	CODE_START := CODE_START + 1;
	// pull out the parameters
	SCREW_PARAMETERS[NS_PITCH] := STRING_TO_REAL(MID(GPS_PNEZD_D, 3, CODE_START));
	SCREW_PARAMS_CUSTOM[0].NS_PITCH := STRING_TO_SINT(MID(GPS_PNEZD_D, 3, CODE_START));
	CODE_START := CODE_START + 3;
	SCREW_PARAMETERS[SCREW_LENGTH] := STRING_TO_REAL(MID(GPS_PNEZD_D, 3, CODE_START));
	SCREW_PARAMS_CUSTOM[0].SCREW_LENGTH := STRING_TO_UINT(MID(GPS_PNEZD_D, 3, CODE_START));
	CODE_START := CODE_START + 3;
	SCREW_PARAMETERS[TRUSS_VERT_ANGLE] := STRING_TO_REAL(MID(GPS_PNEZD_D, 2, CODE_START));
	SCREW_PARAMS_CUSTOM[0].TRUSS_VERT_ANGLE := STRING_TO_USINT(MID(GPS_PNEZD_D, 2, CODE_START));
	CODE_START := CODE_START + 2;
	IF MID(GPS_PNEZD_D, 2, CODE_START) = 'ZZ' OR MID(GPS_PNEZD_D, 2, CODE_START) = 'zz' THEN
		SCREW_PARAMETERS[THIRD_LEG_VERT_ANGLE] := NA;
		SCREW_PARAMS_CUSTOM[0].THIRD_LEG_VERT_ANGLE := TO_USINT(NA);
	ELSE
		SCREW_PARAMETERS[THIRD_LEG_VERT_ANGLE] := STRING_TO_REAL(MID(GPS_PNEZD_D, 2, CODE_START));
		SCREW_PARAMS_CUSTOM[0].THIRD_LEG_VERT_ANGLE := STRING_TO_USINT(MID(GPS_PNEZD_D, 2, CODE_START));
	END_IF
	CODE_START := CODE_START + 2;
	SCREW_PARAMETERS[EMBED_LENGTH] := STRING_TO_REAL(MID(GPS_PNEZD_D, 3, CODE_START));
	SCREW_PARAMS_CUSTOM[0].EMBED_LENGTH := STRING_TO_USINT(MID(GPS_PNEZD_D, 3, CODE_START));
	CODE_START := CODE_START + 3;
	IF MID(GPS_PNEZD_D, 2, CODE_START) = 'ZZ' OR MID(GPS_PNEZD_D, 2, CODE_START) = 'zz' THEN
		SCREW_PARAMETERS[IE_MIN_HAMMER] := NA;
		SCREW_PARAMS_CUSTOM[0].IE_MIN_HAMMER := TO_USINT(NA);
	ELSE
		SCREW_PARAMETERS[IE_MIN_HAMMER] := STRING_TO_REAL(MID(GPS_PNEZD_D, 2, CODE_START));
		SCREW_PARAMS_CUSTOM[0].IE_MIN_HAMMER := STRING_TO_USINT(MID(GPS_PNEZD_D, 2, CODE_START));
	END_IF
	CODE_START := CODE_START + 2;
	IF MID(GPS_PNEZD_D, 2, CODE_START) = 'ZZ' OR MID(GPS_PNEZD_D, 2, CODE_START) = 'zz' THEN
		SCREW_PARAMETERS[IE_MIN_EMBED] := NA;
		SCREW_PARAMS_CUSTOM[0].IE_MIN_EMBED := TO_USINT(NA);
	ELSE
		SCREW_PARAMETERS[IE_MIN_EMBED] := STRING_TO_REAL(MID(GPS_PNEZD_D, 2, CODE_START));
		SCREW_PARAMS_CUSTOM[0].IE_MIN_EMBED := STRING_TO_USINT(MID(GPS_PNEZD_D, 2, CODE_START));
	END_IF
	CODE_START := CODE_START + 2;
	DecodePnezD := TRUE;
	//SCREW_PARAMETERS[TRUSS_TYPE] := AsciiToReal(MID(GPS_PNEZD_D, 1, CODE_START));
	(*
	IF MID(GPS_PNEZD_D, 1, CODE_START) = TRUSS_CODES[] OR MID(GPS_PNEZD_D, 1, CODE_START) = 'i' THEN
		SCREW_PARAMETERS[TRUSS_TYPE] := 0;
	ELSIF MID(GPS_PNEZD_D, 1, CODE_START) = 'E' OR MID(GPS_PNEZD_D, 1, CODE_START) = 'e' THEN
		SCREW_PARAMETERS[TRUSS_TYPE] := 2;
	ELSIF MID(GPS_PNEZD_D, 1, CODE_START) = 'C' OR MID(GPS_PNEZD_D, 1, CODE_START) = 'c' THEN
		SCREW_PARAMETERS[TRUSS_TYPE] := 1;
	ELSE
		DecodePnezD := FALSE;
	END_IF*)

END_FUNCTION

// StandardPLC/Application/POUs/Utilities/Conversions/AsciiToReal
FUNCTION AsciiToReal : REAL
VAR_INPUT
	CHAR: STRING(1);
END_VAR
VAR
	pBYTE: POINTER TO BYTE;
END_VAR

pBYTE := ADR(CHAR);
AsciiToReal := pBYTE^;

END_FUNCTION

// StandardPLC/Application/POUs/Test_PRGs/DynamicList
(* This list self-populates with new values until the max size is reached.
eg, if a new screw size is added, it will automatically add it to the list and start counting that size screw.
*)

PROGRAM DynamicList 
VAR
	// function vars
	i: USINT := 0;
	
	// sim vars
	init: BOOL := TRUE;
	pnezDlast: STRING(64) := '';
	// system vars
	SCREW_COUNT_ORDER: ARRAY [1..SCREW_LENGTHS_COUNT] OF UDINT := [SCREW_LENGTHS_COUNT(0)];
	
	
END_VAR

IF init OR (pnezDlast <> GPS_PNEZD_D) THEN
	init := FALSE;
	pnezDlast := GPS_PNEZD_D;
	
	FOR i := 1 TO SCREW_LENGTHS_COUNT DO
		IF TO_UINT(SCREW_COUNT[1,i]) = TO_UINT(SCREW_PARAMETERS[SCREW_LENGTH]) THEN
			SCREW_COUNT[2,i] := SCREW_COUNT[2,i] + 1;
			EXIT;
		ELSIF TO_UINT(SCREW_COUNT[1,i]) = 0 THEN
			SCREW_COUNT[1,i] := TO_UINT(SCREW_PARAMETERS[SCREW_LENGTH]);
			SCREW_COUNT[2,i] := 1;
			// *** organize list
			WHILE i > 1 DO
				IF SCREW_COUNT[1,i] < SCREW_COUNT[1,i - 1] THEN
					SCREW_COUNT[1,i] := SCREW_COUNT[1,i - 1];
					SCREW_COUNT[2,i] := SCREW_COUNT[2,i - 1];
					SCREW_COUNT[1,i-1] := TO_UINT(SCREW_PARAMETERS[SCREW_LENGTH]);
					SCREW_COUNT[2,i-1] := 1;
				END_IF
				i := i - 1;
			END_WHILE
			EXIT;
			// ^^^
		END_IF
	END_FOR	
END_IF

END_PROGRAM

// StandardPLC/Application/POUs/Test_PRGs/Arrays
PROGRAM Arrays
VAR
	Init: BOOL := TRUE;
	TEST_1: ARRAY [0..20] OF UINT := [15,20(0)]; // first position indicates number of used slots
	TEST_2: ARRAY [3..9] OF BOOL := [7(0)];	
	TEST_3: ARRAY [0..20] OF UINT := [21(0)];
	LOWER_BOUND_TEST_1: USINT := 0;
	LOWER_BOUND_TEST_2: USINT := 0;
	UPPER_BOUND_TEST_1: USINT := 0;
	UPPER_BOUND_TEST_2: USINT := 0;
	LENGTH_TEST_1: USINT := 0;
	LENGTH_TEST_2: USINT := 0;
	SIZE_OF_TEST_1: UINT := 0;
	SIZE_OF_TEST_2: UINT := 0;
	i: UINT := 0;
	j: UINT := 0;
	Timeout_Index: UINT := 0;
END_VAR

IF Init THEN
	Init := FALSE;
	Timeout_Index := 1;
	//LOWER_BOUND_TEST_1 := TO_USINT(LOWER_BOUND(TEST_1, 2));
	//LOWER_BOUND_TEST_2 := TO_USINT(LOWER_BOUND(TEST_2, 1));
	//UPPER_BOUND_TEST_1 := TO_USINT(UpperBoundBool(TEST_1));
	UPPER_BOUND_TEST_2 := TO_USINT(UpperBoundBool(TEST_2));
	SIZE_OF_TEST_1 := SIZEOF(TEST_1);
	SIZE_OF_TEST_2 := SIZEOF(TEST_2);

END_IF
Timeout_Index := Timeout_Index + 1;
IF Timeout_Index <= 200 THEN
	FOR i := 1 TO TEST_1[0] DO
		TEST_1[i] := TEST_1[i] + i;
	END_FOR
ELSIF Timeout_Index = 300 THEN
	TEST_3 := TEST_1;
	
END_IF

END_PROGRAM

// StandardPLC/Application/POUs/Utilities/UpperBoundBool
FUNCTION UpperBoundBool : UINT
VAR_IN_OUT
	INPUT_ARRAY : ARRAY[*] OF BOOL;
END_VAR
VAR_INPUT
	
END_VAR
VAR
END_VAR

UpperBoundBool := TO_UINT(UPPER_BOUND(INPUT_ARRAY, 1));

END_FUNCTION

// Project Information/GetCompany
// This function has been automatically generated from the project information.
{attribute 'signature_flag' := '1073741824'}
{attribute 'register_in_runtime'}
FUNCTION GetCompany : WSTRING
VAR_INPUT
	
END_VAR

GetCompany := "ifm electronic";

END_FUNCTION

// Project Information/GetTitle
// This function has been automatically generated from the project information.
{attribute 'signature_flag' := '1073741824'}
{attribute 'register_in_runtime'}
FUNCTION GetTitle : WSTRING
VAR_INPUT
	
END_VAR

GetTitle := "ifmCR711S_TemplateProject";

END_FUNCTION

// Project Information/GetVersion
// This function has been automatically generated from the project information.
{attribute 'signature_flag' := '1073741824'}
{attribute 'register_in_runtime'}
FUNCTION GetVersion : VERSION
VAR_INPUT
	
END_VAR

GetVersion.uiMajor := 2;
GetVersion.uiMinor := 4;
GetVersion.uiServicePack := 15;
GetVersion.uiPatch := 0;

END_FUNCTION

// Project Information/GetTextProperty
// This function has been automatically generated from the project information.
{attribute 'signature_flag' := '1073741824'}
{attribute 'register_in_runtime'}
FUNCTION GetTextProperty : WSTRING
VAR_INPUT
	stKey: WSTRING;
END_VAR

IF stKey = "Company" THEN
	GetTextProperty := "ifm electronic";
ELSIF stKey = "Description" THEN
	GetTextProperty := "Project template with CR711S configured 2.25MByte Standard 2.25MByte Safety";
ELSIF stKey = "Project" THEN
	GetTextProperty := "experiment_with_CoDeSys_sp16";
ELSIF stKey = "Title" THEN
	GetTextProperty := "ifmCR711S_TemplateProject";
ELSE
	GetTextProperty := "";
END_IF

END_FUNCTION

// Project Information/GetTextProperty2
// This function has been automatically generated from the project information.
{attribute 'signature_flag' := '1073741824'}
{attribute 'register_in_runtime'}
FUNCTION GetTextProperty2 : POINTER TO WSTRING
VAR_INPUT
	stKey: WSTRING;
END_VAR

IF stKey = "Company" THEN
	GetTextProperty2 := ADR("ifm electronic");
ELSIF stKey = "Description" THEN
	GetTextProperty2 := ADR("Project template with CR711S configured 2.25MByte Standard 2.25MByte Safety");
ELSIF stKey = "Project" THEN
	GetTextProperty2 := ADR("experiment_with_CoDeSys_sp16");
ELSIF stKey = "Title" THEN
	GetTextProperty2 := ADR("ifmCR711S_TemplateProject");
ELSE
	GetTextProperty2 := ADR("");
END_IF

END_FUNCTION

// Project Information/GetNumberProperty
// This function has been automatically generated from the project information.
{attribute 'signature_flag' := '1073741824'}
{attribute 'register_in_runtime'}
FUNCTION GetNumberProperty : DINT
VAR_INPUT
	stKey: WSTRING;
END_VAR

GetNumberProperty := 0;

END_FUNCTION

// Project Information/GetBooleanProperty
// This function has been automatically generated from the project information.
{attribute 'signature_flag' := '1073741824'}
{attribute 'register_in_runtime'}
FUNCTION GetBooleanProperty : BOOL
VAR_INPUT
	stKey: WSTRING;
END_VAR

IF stKey = "Released" THEN
	GetBooleanProperty := FALSE;
ELSE
	GetBooleanProperty := FALSE;
END_IF

END_FUNCTION

// Project Information/GetVersionProperty
// This function has been automatically generated from the project information.
{attribute 'signature_flag' := '1073741824'}
{attribute 'register_in_runtime'}
FUNCTION GetVersionProperty : VERSION
VAR_INPUT
	stKey: WSTRING;
END_VAR

IF stKey = "Version" THEN
	GetVersionProperty.uiMajor := 2;
	GetVersionProperty.uiMinor := 4;
	GetVersionProperty.uiServicePack := 15;
	GetVersionProperty.uiPatch := 0;
ELSE
	GetVersionProperty.uiMajor := 0;
	GetVersionProperty.uiMinor := 0;
	GetVersionProperty.uiServicePack := 0;
	GetVersionProperty.uiPatch := 0;
END_IF

END_FUNCTION

// StandardPLC/Application/POUs/Utilities/Conversions/pSQR
FUNCTION pSqr : POINTER TO REAL
VAR_INPUT
	Num: REAL;
	
END_VAR
VAR
		SqrVal: LREAL;
END_VAR


SqrVal := EXPT(Num, 2);
pSqr := ADR (SqrVal);

END_FUNCTION

// StandardPLC/Application/POUs/Utilities/Conversions/SqrReals
FUNCTION SqrReals : REAL
VAR_INPUT
	Num: REAL;

END_VAR
VAR
END_VAR

SqrReals := to_real(EXPT(Num,2));

END_FUNCTION

// StandardPLC/Application/POUs/ConvertDiag
FUNCTION_BLOCK ConvertDiag
VAR_INPUT
	ifmDiag: ifmTYPES.DIAG_INFO;
END_VAR
VAR_OUTPUT
	s_Diag: STRING;
END_VAR
VAR
	i_Diag: Diag;
END_VAR

(* input is TO_INT(ifm ediag's name)
create a diag enum with this as the number
convert diag to string with to_string*)

i_Diag := TO_INT(ifmDiag);
s_Diag := TO_STRING(i_Diag);

END_FUNCTION_BLOCK

// StandardPLC/Application/POUs/ConvDiag
FUNCTION ConvDiag : STRING
VAR_INPUT
		ifmDiag: ifmTYPES.DIAG_INFO;
END_VAR
VAR
	i_diag: diag;
END_VAR



i_diag := TO_INT(ifmDiag);
ConvDiag := TO_STRING(i_diag);

END_FUNCTION

// StandardPLC/Application/POUs/Checksum
FUNCTION Checksum : UINT

VAR_INPUT
	FILE_PTR: POINTER TO BYTE; // pointer to beginning of memory block/file to be checked
	FILE_LENGTH: UINT; // # of bytes in file
END_VAR

VAR
	INDEX: INT; // loop index
	SUM: UINT := 0; // sum of 1's in file
	
END_VAR

FILE_LENGTH := MAX(1,FILE_LENGTH);

FOR INDEX := 1 TO TO_INT(FILE_LENGTH) DO
	SUM := SUM + TO_UINT(FILE_PTR^);
	FILE_PTR := FILE_PTR + 1;
END_FOR

Checksum := SUM;

END_FUNCTION

// StandardPLC/Application/POUs/Utilities/MemBlockLength
FUNCTION MemBlockLength : UINT
VAR_INPUT
	PTR_START: POINTER TO BYTE;
	PTR_END: POINTER TO BYTE;
	
END_VAR
VAR
	FILE_LENGTH: DWORD := 0;
END_VAR


FILE_LENGTH := MAX(1, ABS(PTR_END - PTR_START));
MemBlockLength := TO_UINT(FILE_LENGTH);

END_FUNCTION

// StandardPLC/Application/POUs/Checksum_wLength
FUNCTION Checksum_wLength : UINT

VAR_INPUT
	FILE_BEGIN_PTR: POINTER TO BYTE; // pointer to beginning of memory block/file to be checked
	FILE_END_PTR: POINTER TO BYTE; // pointer to end of memory block/file to be checked
END_VAR

VAR
	INDEX: INT := 0; // loop index
	SUM: UINT := 0; // sum of 1's in file
	
	FILE_LENGTH: UINT := 0;
END_VAR


FILE_LENGTH := MemBlockLength(FILE_BEGIN_PTR, FILE_END_PTR);
FILE_LENGTH := MAX(1,FILE_LENGTH);

FOR INDEX := 1 TO TO_INT(FILE_LENGTH) DO
	SUM := SUM + TO_UINT(FILE_BEGIN_PTR^);
	FILE_BEGIN_PTR := FILE_BEGIN_PTR + 1;
END_FOR

Checksum_wLength := SUM;

END_FUNCTION

// StandardPLC/Application/POUs/Utilities/Conversions/ArrayOfBytesToLWORD
FUNCTION ArrayOfBytesToLWORD : LWORD // not tested
VAR_INPUT
	ARRAY_SIZE: INT :=4; // accept arrays of 2 - 8 BYTES
	LITTLE_ENDIAN: BOOL := TRUE;
END_VAR
VAR_IN_OUT
	BYTE_ARRAY: ARRAY [*] OF BYTE;
END_VAR
VAR
	i: INT :=0;
	dataLWORD: LWORD :=0;
	BArray: ARRAY [0..8] OF BYTE := [0,0,0,0,0,0,0,0];
	
END_VAR

// concat array of bytes into LWORD
// rearrange for endianness
IF LITTLE_ENDIAN THEN
	dataLWORD :=  SHL(TO_LWORD(BArray[0]),8) OR BArray[1];
	FOR i := 0 TO ARRAY_SIZE - 1 DO
		BArray[ARRAY_SIZE - i - 1] := BYTE_ARRAY[i];
	END_FOR
ELSE
	dataLWORD := BArray[1] OR SHL(TO_LWORD(BArray[0]),8);
	FOR i := 0 TO ARRAY_SIZE - 1 DO
		BArray[i] := BYTE_ARRAY[i];
	END_FOR
END_IF

// pack arranged array into LWORD
dataLWORD :=  SHL(TO_LWORD(BArray[0]),8) OR BArray[1];
IF ARRAY_SIZE > 2 THEN
	FOR i := 2 TO ARRAY_SIZE - 1 DO
		dataLWORD := SHL(dataLWORD,8) OR BArray[i];
	END_FOR
END_IF

ArrayOfBytesToLWORD := dataLWORD;

END_FUNCTION

// StandardPLC/Application/POUs/Utilities/Conversions/ConvLWORDtoDecimal
FUNCTION ConvLWORDtoDecimal : REAL
VAR_INPUT
	BINARY: LWORD :=0;
	SCALE: REAL :=0;
	OFFSET: REAL :=0;
END_VAR
VAR
	DEC: INT := 0;
END_VAR

// input LWORD and output the scaled and offset decimal
//DEC := LWORD_TO_REAL (BINARY); // convert to INT first?
DEC := LWORD_TO_INT (BINARY);
ConvLWORDtoDecimal := INT_TO_REAL(DEC) * SCALE + OFFSET;

END_FUNCTION

// StandardPLC/Application/POUs/IsExtendedCAN
FUNCTION IsExtendedCAN : BOOL

VAR_INPUT
	MSG_ID: UDINT;
END_VAR
VAR
END_VAR

//IsExtendedCAN := (MSG_ID > 2047);

IsExtendedCAN := (len(TO_WORD(MSG_ID)) < 12);

END_FUNCTION

// StandardPLC/Application/POUs/getElapsedTime
FUNCTION_BLOCK getElapsedTime // not functional - just recorded ideas, didn't finish
VAR_INPUT
END_VAR
VAR_OUTPUT
END_VAR
VAR
	START: SysTime := 0;
	FINISH: SysTime := 0;
	INTERVAL: SysTime :=0;
	INTERVAL_SUM: SysTime :=0;
	INTERVAL_AVG: SysTime :=0;
END_VAR

// use systime to get microseconds or even nanoseconds for an event

SysTimeGetUs(START); // this is in the SysTime library; optional SysTimeGetNs.  assigns value to supplied variable 
// event occurs
SysTimeGetUs(FINISH);
INTERVAL := FINISH - START;

// if want to get an average add a count something like this:
(*
INTERVAL_SUM := INTERVAL_SUM + INTERVAL;
IF (COUNT MOD 1000 = 0) THEN
	INTERVAL_AVG := INTERVAL_SUM/1000;
	INTERVAL_SUM := 0;
END_IF
*)

END_FUNCTION_BLOCK

// StandardPLC/Application/POUs/Utilities/Conversions/REAL_TO_BYTE_ARRAY
FUNCTION_BLOCK REAL_TO_BYTE_ARRAY // take in a REAL and output an array of bytes
VAR_INPUT
END_VAR
VAR_OUTPUT
END_VAR
VAR
END_VAR

END_FUNCTION_BLOCK

// StandardPLC/Application/POUs/Utilities/Conversions/ArrayOfUsintsToLWORD
FUNCTION ArrayOfUsintsToLWORD : LWORD // not tested, may be a problem with this that crashes PLC
VAR_INPUT
	ARRAY_SIZE: INT :=4; // accept arrays of 2 - 8 BYTES
	LITTLE_ENDIAN: BOOL := TRUE;
END_VAR
VAR_IN_OUT
	BYTE_ARRAY: ARRAY [*] OF USINT;
END_VAR
VAR
	i: INT :=0;
	dataLWORD: LWORD :=0;
	BArray: ARRAY [0..8] OF BYTE := [0,0,0,0,0,0,0,0];
	
END_VAR

// concat array of bytes into LWORD
// rearrange for endianness

IF LITTLE_ENDIAN THEN
	dataLWORD :=  SHL(TO_LWORD(BArray[0]),8) OR BArray[1];
	FOR i := 0 TO ARRAY_SIZE - 1 DO
		BArray[ARRAY_SIZE - i - 1] := TO_BYTE(BYTE_ARRAY[i]);
	END_FOR
ELSE
	dataLWORD := BArray[1] OR SHL(TO_LWORD(BArray[0]),8);
	FOR i := 0 TO ARRAY_SIZE - 1 DO
		BArray[i] := TO_BYTE(BYTE_ARRAY[i]);
	END_FOR
END_IF

// pack arranged array into LWORD
dataLWORD :=  SHL(TO_LWORD(BArray[0]),8) OR BArray[1];
IF ARRAY_SIZE > 2 THEN
	FOR i := 2 TO ARRAY_SIZE - 1 DO
		dataLWORD := SHL(dataLWORD,8) OR BArray[i];
	END_FOR
END_IF

ArrayOfUsintsToLWORD := dataLWORD;

END_FUNCTION

// StandardPLC/Application/POUs/Utilities/Conversions/TAN_DEG
FUNCTION TAN_DEG : REAL
VAR_INPUT
	DEGREES: REAL;
END_VAR
VAR
	RADIANS: REAL;
END_VAR


RADIANS := (3.14159 * DEGREES / 180.0);
TAN_DEG := TAN(RADIANS);

END_FUNCTION

// StandardPLC/Application/POUs/Utilities/ProfileGen/ProfileGenerator_2d
FUNCTION ProfileGenerator_2d
VAR_INPUT
	CURVE_TYPE: INT;// type of curve (linear: -x*var; inverse: x/var; exponential: var^x or var^1/x; log: log x(var); ln: ln(x); sigmoid: [(var-x)/(sqrt(1+(var-x)2] + 1;  ... ?)
	CHAR_VAR: REAL; // characteristic variable (x from above)
	// 2d array of appropriate size
	IND_VAR_LOW: REAL; // independent variable start
	IND_VAR_HIGH: REAL; // independent variable end
	// number of data points desired
	
END_VAR
VAR_IN_OUT
	DATA_ARRAY_X: ARRAY [*] OF REAL; // independent var
	DATA_ARRAY_Y: ARRAY [*] OF REAL; // dependent var
END_VAR
VAR_OUTPUT
END_VAR
VAR
	// dependent variable
	ARRAY_LENGTH: DINT := 1; // number of data points
	i: DINT := 0;
	j: DINT := 0;
END_VAR


ARRAY_LENGTH := UPPER_BOUND(DATA_ARRAY_X,1) - LOWER_BOUND(DATA_ARRAY_X,1) + 1;
DATA_ARRAY_X[1] := IND_VAR_LOW;
IF ARRAY_LENGTH > 1 THEN
	FOR i := 2 TO ARRAY_LENGTH DO
		DATA_ARRAY_X[i] := (IND_VAR_HIGH-IND_VAR_LOW)/(TO_REAL(ARRAY_LENGTH)-1)+DATA_ARRAY_X[i-1];
	END_FOR
	
	FOR i := 1 TO ARRAY_LENGTH DO
		DATA_ARRAY_Y[i] := CurveGenerator_2d(CURVE_TYPE, DATA_ARRAY_X[i], CHAR_VAR);
	END_FOR
END_IF

(*
FOR i := LOWER_BOUND(DATA_ARRAY,1) TO UPPER_BOUND(DATA_ARRAY,1) 
	DATA_ARRAY[
END_FOR
// *)

END_FUNCTION

// StandardPLC/Application/POUs/Utilities/ProfileGen/CurveGenerator_2d
FUNCTION CurveGenerator_2d : REAL
VAR_INPUT
	CURVE_TYPE: INT;// type of curve (linear: x*var; inverse: x/var; exponential: var^x or var^1/x; log: log x(var); ln: ln(x); sigmoid: [(var-x)/(sqrt(1+(var-x)2] + 1;  ... ?)
	IND_VAR: REAL;// ind var
	CHAR_VAR: REAL; // characteristic variable (x from above)
	
END_VAR
VAR
END_VAR



CASE CURVE_TYPE OF
	1: CurveGenerator_2d := CHAR_VAR * IND_VAR; // linear
	2: CurveGenerator_2d := CHAR_VAR/IND_VAR; // inverse
	3: CurveGenerator_2d := EXPT(IND_VAR, CHAR_VAR); // exponent
	4: CurveGenerator_2d := EXPT(CHAR_VAR, IND_VAR); // exponential
	5: CurveGenerator_2d := CHAR_VAR*LOG(IND_VAR); // log
	6: CurveGenerator_2d := CHAR_VAR*LN(IND_VAR); // ln
	7: CurveGenerator_2d := ((IND_VAR - CHAR_VAR)/SQRT(1+EXPT((IND_VAR-CHAR_VAR),2))) + 1; // sigmoid
	8: CurveGenerator_2d :=  IND_VAR; // 
	9: CurveGenerator_2d :=  IND_VAR; // 
	10: CurveGenerator_2d :=  IND_VAR; // 
END_CASE
(*  Can't use enums for CASE??
CASE CURVE_TYPE OF
	LINEAR:  CurveGenerator_2d := CHAR_VAR * IND_VAR; // linear
	INVERSE: CurveGenerator_2d := CHAR_VAR/IND_VAR; // inverse
	EXPONENTIAL: CurveGenerator_2d := IND_VAR^CHAR_VAR; // exponential
	LOGB10: CHAR_VAR*LOG(IND_VAR); // log
	NATLOG: CHAR_VAR*LN(IND_VAR); // ln
	SIGMOID:
	RES1: 
	RES2: 
	RES3:
END_CASE

//*)

END_FUNCTION

// StandardPLC/Application/POUs/Utilities/ProfileGen/TDcontrolCode/setVelAccel
FUNCTION setVelAccel : BOOL 
	(* Use this to have an axis try to continuously settle to a setpoint when the actual
		position is disturbed by external forces, for instance on these axes:
		
			1) Pitch (by tracks moving across uneven ground)
			2) Rotator (by tracks moving across uneven ground)
			3) Yaw pointed to off-machine target (by boom swing moving underneath the yaw)
			
		This function puts a poor-mans motion profile on this action, mainly by controlling the Vff term
			of the loop.  You pass this function the maximum closing velocity for the axis, and the maximum
			acceleration, to control this element, and a position error range for which to feather from 0 velocity
			to some maximum velocity.
			
		The output of this function should be used as input to a PID loop with Vff.
		
		eMax MUST be > eMin or get divide by zero error!
	*)
VAR_INPUT
	(* Desired final position, engr. *)
	TARGET: REAL;
	(* Current position, engr. *)
	ACTUAL: REAL;
	(* Error at which maximum velocity is used, engr. *)
	EMAX: REAL;
	(* Error below which 0 velocity is used, so integrator will mostly close this error, engr. *)
	EMIN: REAL;
	(* Maximum desired velocity, engr. *)
	VMAX: REAL;
	(* Maximum desired acceleration, engr. *)
	AMAX: REAL;
	(* Desired velocity at the current position error, engr. *)
	pVEL: POINTER TO REAL;
	(* Desired acceleration at the current position error, engr. *)
	pACCEL: POINTER TO REAL;
END_VAR
VAR
	ERROR: REAL;
	ERROR_ABS: REAL;
END_VAR


	ERROR := TARGET - ACTUAL;
	ERROR_ABS := ABS(ERROR);
	IF ERROR_ABS > EMAX THEN
		pACCEL^ := AMAX;
		pVEL^ := VMAX;
	ELSIF ERROR_ABS > EMIN THEN
		pACCEL^ := AMAX;
		pVEL^ := VMAX * (ERROR_ABS - EMIN) / (EMAX - EMIN);
	ELSE
		pACCEL^ := 0;
		pVEL^ := 0;
	END_IF

	IF ERROR < 0 THEN
		pACCEL^ := -pACCEL^;
		pVEL^ := -pVEL^;
	END_IF

END_FUNCTION

// StandardPLC/Application/POUs/Utilities/ProfileGen/SetpointInit
FUNCTION SetpointInit : BOOL
VAR_INPUT
	pSETPOINT: POINTER TO sSetpoint;
	FB: sFeedback;
	POS: REAL;
	VEL: REAL;
	ACCEL: REAL;

END_VAR
VAR
END_VAR

pSETPOINT^.POSITION_ENGR := POS;
pSETPOINT^.VELOCITY_ENGR := VEL;
pSETPOINT^.ACCELERATION_ENGR := ACCEL;

pSETPOINT^.POSITION_RAW := POS_ENGR_TO_RAW(FB, POS);
pSETPOINT^.VELOCITY_RAW := VEL_ENGR_TO_RAW(FB, VEL);
pSETPOINT^.ACCELERATION_RAW := VEL_ENGR_TO_RAW(FB, ACCEL);

pSETPOINT^.SETPOINT_CHANGED := TRUE;

SetpointInit := TRUE;

END_FUNCTION

// StandardPLC/Application/POUs/Utilities/ProfileGen/TDcontrolCode/POS_ENGR_TO_RAW
(* Function to convert a number in engineering units to the raw encoder counts that represents the same position. *)
FUNCTION POS_ENGR_TO_RAW : DINT
VAR_INPUT
	FB: sFeedback;
	ENGR: REAL;
END_VAR
VAR
END_VAR


POS_ENGR_TO_RAW := TO_DINT(ENGR * FB.RAW_PER_ENGR);

END_FUNCTION

// StandardPLC/Application/POUs/Utilities/ProfileGen/TDcontrolCode/VEL_ENGR_TO_RAW
FUNCTION VEL_ENGR_TO_RAW : REAL
VAR_INPUT
	FB: sFeedback;
	VEL_OR_ACCEL: REAL;END_VAR
VAR
END_VAR

VEL_ENGR_TO_RAW := VEL_OR_ACCEL * FB.RAW_PER_ENGR;

END_FUNCTION

// StandardPLC/Application/POUs/Utilities/ProfileGen/TDcontrolCode/FeedbackInit
FUNCTION FeedbackInit : BOOL
VAR_INPUT
	pFEEDBACK: POINTER TO sFeedback;

	(* This is the counts of the feedback per engineering unit on the axis. *)
	RAW_PER_ENGR : REAL;
	(* This is the counts on the feedback when the axis is at the position you want
		to call 0 in engineering units. *)
	RAW_WHEN_ENGR_ZERO: UDINT;

	(* Maximium valid feedback reading, in engineering units.  This should be far
		enough past the maximum command limit to tolerate the maximum expected overshoot
		when settling. *)
	FB_VALID_MAX: REAL;
	(* Minimum valid feedback reading, in engineering units.  This should be far
		enough past the minimum command limit to tolerate the maxium expected overshoot
		when settling. *)
	FB_VALID_MIN: REAL;

	(* *)
	ROLLOVER_AT: DINT;
END_VAR
VAR
END_VAR

pFEEDBACK^.RAW_PER_ENGR := RAW_PER_ENGR;

pFEEDBACK^.FEEDBACK_VALID_MAX := POS_ENGR_TO_RAW(pFEEDBACK^, FB_VALID_MAX);
pFEEDBACK^.FEEDBACK_VALID_MIN := POS_ENGR_TO_RAW(pFEEDBACK^, FB_VALID_MIN);

pFEEDBACK^.ROLLOVER_AT := ROLLOVER_AT;
pFEEDBACK^.ROLLOVER_HALF := ROLLOVER_AT / 2;

//AxisZeroInit(pFEEDBACK := pFEEDBACK, RAW_WHEN_ENGR_ZERO := RAW_WHEN_ENGR_ZERO);

(* Now reset dynamic information, especially important on single turn encoders that have to handle rollover. *)
pFEEDBACK^.US_LAST_SAMPLE := 0;
pFEEDBACK^.COUNT := 0;

END_FUNCTION

// StandardPLC/Application/POUs/Utilities/Conversions/CanMsgIdToNodeIndexSubIndex
FUNCTION CanMsgIdToNodeIndexSubIndex : usint
VAR_INPUT
	MSG_ID: UDINT;
END_VAR
VAR_OUTPUT
	NODE_ID: USINT;
	SUB_INDEX: USINT;
	INDEX: UINT;
END_VAR
VAR
END_VAR

NODE_ID := TO_USINT(16#FF AND MSG_ID); // pull right 8 bits
SUB_INDEX := to_USINT(SHR(MSG_ID, 8) and 16#FF); // pull next 8 bits
INDEX := to_UINT (SHR(MSG_ID, 16) AND 16#FF); // pull last (left most) 16 bits

END_FUNCTION

// StandardPLC/Application/POUs/Utilities/Conversions/CanNodeIndexSubIndexToJ1939MsgId
FUNCTION CanNodeIndexSubIndexToJ1939MsgId : UDINT
VAR_INPUT
	NODE: USINT;
	SUB_INDEX: USINT;
	INDEX: UDINT;
END_VAR
VAR
END_VAR

CanNodeIndexSubIndexToJ1939MsgId := 16#18000000 + SHL(INDEX, 16) + SHL(SUB_INDEX, 8) + NODE;

END_FUNCTION

// StandardPLC/Application/POUs/Utilities/Conversions/ACOS_DEG
FUNCTION ACOS_DEG: REAL
VAR_INPUT
	VALUE: REAL;
END_VAR
VAR
END_VAR

//ACOS_DEG := (180 * ACOS(VALUE)) / 3.14159;

IF ABS(VALUE) > 1 THEN // prevent killing PLC with a NaN if bad value sent
	VALUE := MAX(MIN(VALUE, -1),1);
END_IF

ACOS_DEG := (180 * ACOS(VALUE)) / Pi;

END_FUNCTION

// StandardPLC/Application/POUs/Utilities/DataSmoothing
FUNCTION_BLOCK DataSmoothing
// take in a data point and x number of points to average, and return a running average of the last x entries

VAR_INPUT
	CURRENT_DATA_POINT: REAL;
	NUM_POINTS_TO_AVERAGE: USINT; //(limit 255, @ 50hz = 5.1 seconds)
END_VAR
VAR_OUTPUT
	SMOOTHED_DATA_OUTPUT: REAL;
END_VAR
VAR
	DATA_POINTS: ARRAY [1..255] OF REAL := [255(0)];
	NUM_OF_COLLECTED_ENTRIES: USINT;
	ENTRY_INDEX: USINT := 1;
	DATA_ARRAY_FULL: BOOL := FALSE;
	DATA_SUM: REAL := 0;
	AVG_INDEX: USINT := 1;
END_VAR

// store sample
DATA_POINTS[ENTRY_INDEX] := CURRENT_DATA_POINT;

// average collected data
DATA_SUM := 0; // clear history
FOR AVG_INDEX := 1 TO NUM_POINTS_TO_AVERAGE DO
	DATA_SUM := DATA_SUM + DATA_POINTS[AVG_INDEX];
END_FOR

IF DATA_ARRAY_FULL THEN
	SMOOTHED_DATA_OUTPUT := DATA_SUM / NUM_POINTS_TO_AVERAGE;
ELSE 
	SMOOTHED_DATA_OUTPUT := DATA_SUM / ENTRY_INDEX;
END_IF

// update entry number
// control how many entries to average (correlates to delay time of averaging)
IF ENTRY_INDEX < NUM_POINTS_TO_AVERAGE THEN
	ENTRY_INDEX := ENTRY_INDEX +1;
ELSE
	ENTRY_INDEX := 1;
	DATA_ARRAY_FULL := TRUE;
END_IF

END_FUNCTION_BLOCK

// StandardPLC/Application/POUs/Utilities/ProfileGen/ScurveProfiler
FUNCTION_BLOCK ScurveProfiler
VAR_INPUT
	TIME_START: DWORD;
	TIME_NOW_US: DWORD;
	CURRENT_POS_ENGR: REAL;
	START_POS_ENGR: REAL;
	END_POS_ENGR: REAL;
	Vmax: REAL;
	Amax: REAL;
END_VAR
VAR_OUTPUT
	STEP_TARGET_POS: REAL;
	STEP_TARGET_VEL: REAL;
	
END_VAR
VAR
	LAST_STEP_POS: REAL;
	MIDPOINT: DWORD := 0;
	T_shift: REAL := 0;
	Afin: REAL := 0;
	MODE: USINT := 0;
	T: REAL := 0;
	Z: REAL := 0;
	STEP_TARGET_VEL_MIDPOINT: REAL := 0;
	Vmove: REAL := 0;
	Amove: REAL := 0;
	INDEX: USINT := 1;
	
END_VAR


(*
return current position based on desired current velocity * time delta
calc current velocity by s-curves
reverse s-curve at halfway point
*)
T_shift := SQRT ( (14 / EXPT(( 1/Amax ),1.5)) - Amax );
Afin := Amax / (0.5 * Vmax);
T := TO_REAL(TIME_NOW_US) - T_shift;
Z := 1 / EXPT(Afin, 2);
// <Need integral to determine if we reach flat part of vel curve>
// integrate 
(*
Take integral
*)

Amove := Amax;
Vmove := Vmax;
WHILE INDEX > 0 DO
	STEP_TARGET_VEL_MIDPOINT := 

	IF  STEP_TARGET_VEL_MIDPOINT > 0.9 * Vmax THEN
		INDEX := 0;
	ELSE 
		
	END_IF
END_WHILE
	
STEP_TARGET_VEL :=  T /( SQRT ( Z + EXPT( T , 2 ) ));
	
(*
V(t) = { [ ( t - t_shift ) / (SQRT ( (1 / (af^2)) + t - t_shift )^2 ) ] +1 } *  ( Vmax / 2 )
T shift = t_shift = SQRT ( ( 14 / (1/z)^⅔) - z )
af = ( a_max ) /(  max vel / 2 )
*)

(*

IF TARGET_POS < 0 THEN
			IF GPS_TARGET_INIT THEN // set initial reference position to calc offsets/cycle from
				TARGET_LAST := AXES[AXIS_YAW].FEEDBACK.POSITION_ENGR;
				GPS_TARGET_INIT := FALSE;
			END_IF
			TARGET_POS := MAX(-1*GPS_LOOP_MAX_VEL + TARGET_LAST, TARGET_POS); // limit position change to control velocity
		ELSE
			IF GPS_TARGET_INIT THEN
				TARGET_LAST := AXES[AXIS_YAW].FEEDBACK.POSITION_ENGR;
				GPS_TARGET_INIT := FALSE;
			END_IF
			TARGET_POS := MIN(GPS_LOOP_MAX_VEL + TARGET_LAST, TARGET_POS);
		END_IF
		TARGET_LAST := TARGET_POS;

*)

END_FUNCTION_BLOCK

// StandardPLC/Application/POUs/Utilities/DataSmoothing_1
FUNCTION_BLOCK DataSmoothing_1
// take in a data point and x number of points to average, and return a running average of the last x entries
// reject crazy outliers

VAR_INPUT
	CURRENT_DATA_POINT: REAL;
	NUM_POINTS_TO_AVERAGE: USINT; //(limit 100, @ 50hz = 2 seconds)
END_VAR
VAR_OUTPUT
	SMOOTHED_DATA_OUTPUT: REAL :=0;
END_VAR
VAR
	DATA_POINTS: ARRAY [1..100] OF REAL := [100(0)];
	NUM_OF_COLLECTED_ENTRIES: USINT;
	ENTRY_INDEX: USINT := 1;
	DATA_ARRAY_FULL: BOOL := FALSE;
	DATA_SUM: REAL := 0;
	AVG_INDEX: USINT := 1;
	LAST_SMOOTHED_DATA_OUTPUT: REAL := 0;
	LAST_DATA_POINT: REAL := 0;
	INIT: BOOL := TRUE;
	DELTA: REAL := 0;
	LAST_DELTA: REAL := 0;
END_VAR


NUM_POINTS_TO_AVERAGE := MAX(1, NUM_POINTS_TO_AVERAGE);


//IF NOT INIT THEN
DELTA := ABS(CURRENT_DATA_POINT - LAST_DATA_POINT);
	//IF CURRENT_DATA_POINT > (5 * LAST_DATA_POINT + 5 * LAST_DELTA) THEN

IF LAST_DELTA <> 0 AND DELTA > ( 10 * LAST_DELTA) THEN 
	CURRENT_DATA_POINT := ( SMOOTHED_DATA_OUTPUT - LAST_SMOOTHED_DATA_OUTPUT ) + LAST_DATA_POINT;
END_IF
LAST_DATA_POINT := CURRENT_DATA_POINT;	
LAST_DELTA := DELTA;	
//END_IF
(*
IF NOT init THEN
	IF ABS(LAST_DATA_POINT) > 0 THEN // exclude first time or 0's ( because anything is > 5*0 )
		IF  ABS(CURRENT_DATA_POINT) > ( 5*ABS(LAST_DATA_POINT) ) THEN
			CURRENT_DATA_POINT := ( SMOOTHED_DATA_OUTPUT - LAST_SMOOTHED_DATA_OUTPUT ) + LAST_DATA_POINT;
		ELSE
			LAST_DATA_POINT := CURRENT_DATA_POINT;	
		END_IF
	
	END_IF
ELSE
	LAST_DATA_POINT := CURRENT_DATA_POINT;
	init := FALSE;
END_IF
*)

LAST_SMOOTHED_DATA_OUTPUT := SMOOTHED_DATA_OUTPUT;

// store sample
DATA_POINTS[ENTRY_INDEX] := CURRENT_DATA_POINT;

// average collected data
DATA_SUM := 0; // clear history
FOR AVG_INDEX := 1 TO NUM_POINTS_TO_AVERAGE DO
	DATA_SUM := DATA_SUM + DATA_POINTS[AVG_INDEX];
END_FOR

IF DATA_ARRAY_FULL THEN
	SMOOTHED_DATA_OUTPUT := DATA_SUM / NUM_POINTS_TO_AVERAGE;
ELSE 
	SMOOTHED_DATA_OUTPUT := DATA_SUM / ENTRY_INDEX;
END_IF

// update entry number
// control how many entries to average (correlates to delay time of averaging)
IF ENTRY_INDEX < NUM_POINTS_TO_AVERAGE THEN
	ENTRY_INDEX := ENTRY_INDEX +1;
ELSE
	ENTRY_INDEX := 1;
	DATA_ARRAY_FULL := TRUE;
END_IF

END_FUNCTION_BLOCK

// StandardPLC/Application/POUs/Utilities/DataSmoothing_2
FUNCTION_BLOCK DataSmoothing_2
// take in a data point and x number of points to average, and return a running average of the last x entries

VAR_INPUT
	CURRENT_DATA_POINT: REAL;
	NUM_POINTS_TO_AVERAGE: UINT; //(limit 255, @ 50hz = 5.1 seconds)
	RANGE_MIN: REAL;
	RANGE_MAX: REAL;
END_VAR
VAR_OUTPUT
	SMOOTHED_DATA_OUTPUT: REAL;
END_VAR
VAR
	DATA_POINTS: ARRAY [1..255] OF REAL := [255(0)];
	NUM_OF_COLLECTED_ENTRIES: UINT;
	ENTRY_INDEX: UINT := 1;
	DATA_ARRAY_FULL: BOOL := FALSE;
	DATA_SUM: REAL := 0;
	AVG_INDEX: UINT := 1;
	LAST_SMOOTHED_DATA_OUTPUT: REAL := 0;
	LAST_DATA_POINT: REAL :=0;
END_VAR


IF CURRENT_DATA_POINT > RANGE_MAX OR CURRENT_DATA_POINT < RANGE_MIN THEN
	CURRENT_DATA_POINT := ( SMOOTHED_DATA_OUTPUT - LAST_SMOOTHED_DATA_OUTPUT ) + LAST_DATA_POINT;
END_IF


// store sample
DATA_POINTS[ENTRY_INDEX] := CURRENT_DATA_POINT;
LAST_SMOOTHED_DATA_OUTPUT := SMOOTHED_DATA_OUTPUT;
LAST_DATA_POINT := CURRENT_DATA_POINT;

// average collected data
DATA_SUM := 0; // clear history
FOR AVG_INDEX := 1 TO NUM_POINTS_TO_AVERAGE DO
	DATA_SUM := DATA_SUM + DATA_POINTS[AVG_INDEX];
END_FOR

IF DATA_ARRAY_FULL THEN
	SMOOTHED_DATA_OUTPUT := DATA_SUM / NUM_POINTS_TO_AVERAGE;
ELSE 
	SMOOTHED_DATA_OUTPUT := DATA_SUM / ENTRY_INDEX;
END_IF

// update entry number
// control how many entries to average (correlates to delay time of averaging)
IF ENTRY_INDEX < NUM_POINTS_TO_AVERAGE THEN
	ENTRY_INDEX := ENTRY_INDEX +1;
ELSE
	ENTRY_INDEX := 1;
	DATA_ARRAY_FULL := TRUE;
END_IF

END_FUNCTION_BLOCK

// StandardPLC/Application/POUs/GPS/GPS_Y_TO_BS_ANGLE_1
FUNCTION GPS_Y_TO_BS_ANGLE_1 : REAL // angle to move BS by to align end of BS with y of target

VAR_INPUT // most of these will be available in TD code
	YAW_ANGLE: REAL; // angle of yaw arm relative to BS per TD
	HEADING_OFFSET_GPS: REAL; // YAW_BEGIN, or heading offset of wp in world; + is moving mast to the right (CCW) of operator
	X_TD_WP: REAL := 0; // offsets from WP given by gps, + is forward of operator 
	Y_TD_WP: REAL := 0; // + is to the right of operator (facing forward at rear [mast end] of TD)
	
END_VAR
VAR
	BS_7_WORLD: REAL; // boom swing angle relative to North
	BS_l: REAL := 135; // length of boom swing arm
	BS_PIVOT_TO_YAW_PIVOT_Y_WORLD: REAL; // Y delta of BS arm in world frame
	BS_ORIGIN_TO_TARGET_Y_DELTA: REAL; // distance in Y from BS origin to target point
	BS_HEADING_OFFSET_TARGET: REAL; // BS angle from pointing North
	Y_DELTA_WORLD: REAL; // y delta in world frame (vs TD frame as given by gps)
	X_DELTA_WORLD: REAL; // not used here except to call function to get Y
END_VAR

// calculate how much we need to move bs by to align end (yaw pivot) with y of target 

// First correct heading (yaw arm aligned N-S
GPS_Y_TO_BS_ANGLE_1 := HEADING_OFFSET_GPS;



GpsTdToWorldFixedYaw( X_TD_WP := X_TD_WP, Y_TD_WP := Y_TD_WP, YAW_BEGIN := HEADING_OFFSET_GPS, X_WORLD_WP => X_DELTA_WORLD, Y_WORLD_WP => Y_DELTA_WORLD);

BS_7_WORLD := -YAW_ANGLE - HEADING_OFFSET_GPS;
BS_PIVOT_TO_YAW_PIVOT_Y_WORLD := SIN_DEG(BS_7_WORLD) * BS_l;
BS_ORIGIN_TO_TARGET_Y_DELTA := BS_PIVOT_TO_YAW_PIVOT_Y_WORLD + Y_DELTA_WORLD;
BS_HEADING_OFFSET_TARGET := ASIN_DEG( BS_ORIGIN_TO_TARGET_Y_DELTA / BS_l );
GPS_Y_TO_BS_ANGLE :=  BS_HEADING_OFFSET_TARGET - BS_7_WORLD ;

END_FUNCTION

// StandardPLC/Application/POUs/GPS/GPS_Y_TO_BS_ANGLE_2
FUNCTION GPS_Y_TO_BS_ANGLE_2 : REAL // angle to move BS by to align end of BS with y of target

VAR_INPUT // most of these will be available in TD code
	YAW_ANGLE: REAL; // angle of yaw arm relative to BS per TD
	HEADING_OFFSET_GPS: REAL; // YAW_BEGIN, or heading offset of wp in world; + is moving mast to the right (CCW) of operator
	X_TD_WP: REAL := 0; // offsets from WP given by gps, + is forward of operator 
	Y_TD_WP: REAL := 0; // + is to the right of operator (facing forward at rear [mast end] of TD)
	
END_VAR
VAR
	BS_7_OFFSET_WORLD: REAL; //  How far boom swing would rotate to align N-S (in terms of bs move - cw is negative)
	BS_l: REAL := 135; // length of boom swing arm
	BS_PIVOT_TO_YAW_PIVOT_Y_WORLD: REAL; // Y delta of BS arm in world frame from bs pivot to yaw pivot
	BS_PIVOT_TO_TARGET_Y_DELTA: REAL; // distance in Y from BS origin (bs pivot) to target point
	BS_PIVOT_TO_TARGET_Y_HEADING: REAL; // BS angle from pointing North
	Y_DELTA_WORLD: REAL; // y delta in world frame (vs TD frame as given by gps)
	X_DELTA_WORLD: REAL; // not used here except to call function to get Y
END_VAR

// calculate how much we need to move bs by to align end (yaw pivot) with y of target 

GpsTdToWorldFixedYaw( X_TD_WP := X_TD_WP, Y_TD_WP := Y_TD_WP, YAW_BEGIN := HEADING_OFFSET_GPS, X_WORLD_WP => X_DELTA_WORLD, Y_WORLD_WP => Y_DELTA_WORLD);

BS_7_OFFSET_WORLD := - YAW_ANGLE + HEADING_OFFSET_GPS;
BS_PIVOT_TO_YAW_PIVOT_Y_WORLD := -SIN_DEG(BS_7_OFFSET_WORLD) * BS_l;
BS_PIVOT_TO_TARGET_Y_DELTA := BS_PIVOT_TO_YAW_PIVOT_Y_WORLD + Y_DELTA_WORLD;
IF ABS(BS_PIVOT_TO_TARGET_Y_DELTA) > BS_l THEN
	BS_PIVOT_TO_TARGET_Y_HEADING := BS_7_OFFSET_WORLD;
ELSE
	BS_PIVOT_TO_TARGET_Y_HEADING := ASIN_DEG( BS_PIVOT_TO_TARGET_Y_DELTA / BS_l );
END_IF

GPS_Y_TO_BS_ANGLE :=  -(BS_PIVOT_TO_TARGET_Y_HEADING - BS_7_OFFSET_WORLD) ;

END_FUNCTION

// StandardPLC/Application/POUs/GPS/GpsTransform3d
FUNCTION GpsTransform3d : real
VAR_INPUT
END_VAR
VAR
END_VAR

// input x and y before corrections and get x and y values after aligning heading and accounting for pitch and roll

// yaw transform - get x and y

// pitch transform - get x and y

// roll transform - get x and y

// final x and y values

END_FUNCTION

// StandardPLC/Application/POUs/Utilities/ProfileGen/AutotargetIncrementPos
FUNCTION AutotargetIncrementPos : real
VAR_INPUT
	TARGET_POS: REAL;
	TARGET_LAST: REAL; // IF initiating autofeedback move, send current position, else send last targeted position
	VEL: REAL;
END_VAR
VAR
	LOOP_MAX_DELTA_P_PER_CYCLE: REAL;
	
	// testing var's
	CONTROL_FREQ_HZ: REAL := 50;
	
END_VAR


// maps desired max velocity to max position change / cycle
LOOP_MAX_DELTA_P_PER_CYCLE := VEL / CONTROL_FREQ_HZ; // GPS_VEL deg / sec * 0.020 sec / cycle = GPS_LOOP_MAX deg / this cycle
	
IF ABS( TARGET_POS - TARGET_LAST ) > LOOP_MAX_DELTA_P_PER_CYCLE THEN	
	IF ( TARGET_POS - TARGET_LAST ) < 0 THEN // moving in (-) direction
		AutotargetIncrementPos := -1 * LOOP_MAX_DELTA_P_PER_CYCLE + TARGET_LAST; // limit position change to control velocity
	ELSE
		AutotargetIncrementPos := LOOP_MAX_DELTA_P_PER_CYCLE + TARGET_LAST;
	END_IF
ELSE
	AutotargetIncrementPos := TARGET_POS;
END_IF

END_FUNCTION

// StandardPLC/Application/POUs/Utilities/ProfileGen/GpsFeedbackAutotarget
FUNCTION GpsFeedbackAutotarget : REAL

VAR_INPUT
	TARGET_POS: REAL;
	TARGET_LAST: REAL; // IF initiating autofeedback move, send current position, else send last targeted position
	CURRENT_POS: REAL; // current position of actuator 
	GPS_VEL: REAL;
	GPS_ACCEL: REAL;
	GPS_AXIS: USINT;
	GPS_TARGET_INIT: BOOL;
	pAXIS: POINTER TO sAxis;
	(* Desired velocity at the current position error, engr. *)
	pVEL: POINTER TO REAL;
	(* Desired acceleration at the current position error, engr. *)
	pACCEL: POINTER TO REAL;
END_VAR
VAR
	GPS_LOOP_MAX_DELTA_P_PER_CYCLE: REAL;
	TARGET_POS_INCREMENTED: REAL;
	// testing var's
	CONTROL_FREQ_HZ: REAL := 50;
	
END_VAR


		// maps desired max velocity to max position change / cycle
		GPS_LOOP_MAX_DELTA_P_PER_CYCLE := GPS_VEL / CONTROL_FREQ_HZ; // GPS_VEL deg / sec * 0.020 sec / cycle = GPS_LOOP_MAX deg / this cycle
			
		
		IF TARGET_POS < 0 THEN
			IF GPS_TARGET_INIT THEN // set initial reference position to calc offsets/cycle from
				TARGET_LAST := AXES[AXIS_YAW].FEEDBACK.POSITION_ENGR;
				GPS_TARGET_INIT := FALSE;
			END_IF
			TARGET_POS := MAX(-1*GPS_LOOP_MAX_DELTA_P_PER_CYCLE + TARGET_LAST, TARGET_POS); // limit position change to control velocity
		ELSE
			IF GPS_TARGET_INIT THEN
				TARGET_LAST := AXES[AXIS_YAW].FEEDBACK.POSITION_ENGR;
				GPS_TARGET_INIT := FALSE;
			END_IF
			TARGET_POS := MIN(GPS_LOOP_MAX_DELTA_P_PER_CYCLE + TARGET_LAST, TARGET_POS);
		END_IF
		
IF GPS_TARGET_INIT THEN // set initial reference position to calc offsets/cycle from
	TARGET_LAST := pAXIS^.FEEDBACK.POSITION_ENGR;
	GPS_TARGET_INIT := FALSE;
END_IF

IF TARGET_POS < 0 THEN
	GpsFeedbackAutotarget := MAX(-1*GPS_LOOP_MAX_DELTA_P_PER_CYCLE + TARGET_LAST, TARGET_POS); // limit position change to control velocity
ELSE
	GpsFeedbackAutotarget := MIN(GPS_LOOP_MAX_DELTA_P_PER_CYCLE + TARGET_LAST, TARGET_POS);
END_IF
setVelAccel(GpsFeedbackAutotarget, pAXIS^.FEEDBACK.POSITION_ENGR,
	// 3 and 0.1 set to widen deceleration band and approach 0
	3*GPS_AXES[GPS_AXIS].TARGET_LIMIT, 0.01*GPS_AXES[GPS_AXIS].TARGET_LIMIT, GPS_VEL, GPS_ACCEL, pVEL, pACCEL;
SetpointInit(ADR(pAXIS^.SETPOINT), pAXIS^.FEEDBACK, GpsFeedbackAutotarget, pVEL^, pACCEL^);

CLOSED_LOOP := TRUE;	
END_IF

END_FUNCTION

// StandardPLC/Application/POUs/GPS/CheckGpsInRange
PROGRAM CheckGpsInRange
VAR
	
END_VAR

GPS_IN_RANGE := GpsAutotargetInRange(100);

END_PROGRAM

// StandardPLC/Application/POUs/GPS/GpsAutoTrack_1
(* autotrack to gps target

create approach curve by floating target point that moves from 1/3 of distance to target
to 4 m behind target, then align to target and finish drive straignt on
*)
PROGRAM GpsAutoTrack_1
//FUNCTION GpsAutoTrack : BOOL   // autotrack to gps target
VAR_INPUT
	// leave as input in case we want to control to a different point, eg 3rd leg motor
	X_OFFSET_BEGIN: REAL := 0; // offsets from WP given by gps, in TD frame, + is forward of operator 
	Y_OFFSET_BEGIN: REAL := 0; // + is to the right of operator (facing forward at rear [mast end] of TD)
	YAW_OFFSET_BEGIN: REAL := 0; // heading offset to rotate by as given by gps, + is moving mast to the right (CCW) of operator
	Z_OFFSET_BEGIN: REAL := 0; // + is up
END_VAR
VAR_OUTPUT
	LEFT_TRACK_OUTPUT_MAGNITUDE: INT := 0; // send as percent to joystick controller
	RIGHT_TRACK_OUTPUT_MAGNITUDE: INT := 0;
	LEFT_TRACK_OUTPUT_POSITIVE: BOOL := TRUE;
	RIGHT_TRACK_OUTPUT_POSITIVE: BOOL := TRUE;
END_VAR
VAR
	X_OFFSETS: ARRAY [1..9] OF REAL := [9(0)];
	Y_OFFSETS: ARRAY [1..9] OF REAL := [9(0)];
	YAW_OFFSETS: ARRAY [1..9] OF REAL := [9(0)];
	BS_ANGLE_NS_DELTA: REAL := 0;
	BS_ANGLE_WORLD_NS: REAL := 0;
	BS_ANGLE_NS_TO_Y_TARGET_DELTA: REAL := 0;
	YAW_ARM_LENGTH: REAL := 135; // 135 for TD3 with x slide at 0
	//HEADING_TO_TARGET: REAL := 0;
	//LEFT_TRACK_OUTPUT: REAL := 0;
	//RIGHT_TRACK_OUTPUT: REAL := 0;
	LEFT_TRACK_POSITIVE: BOOL := TRUE;
	RIGHT_TRACK_POSITIVE: BOOL := TRUE;
	PROXIMITY_SLOWING_FACTOR: REAL := 1;
	ALIGNMENT_TARGET: REAL := 100; // cm, point before actual target to aim for, then align
	MANUAL_SPEED_REDUCING_FACTOR: REAL := 1;
	GPS_AUTO_TRACK_JOYSTICK_LIMIT: REAL := 70;
	
END_VAR


X_OFFSET_BEGIN := X_OFFSET_BEGIN/10; // convert mm to cm
Y_OFFSET_BEGIN := Y_OFFSET_BEGIN/10; // convert mm to cm
//YAW_OFFSET_BEGIN := YAW_OFFSET_BEGIN; // deg to deg
//Z_OFFSET_BEGIN := Z_OFFSET_BEGIN/10; // convert mm to cm
YAW_ARM_LENGTH := YAW_PIVOT_TO_DRILL_ROD + AXES[AXIS_X_SLIDE].FEEDBACK.POSITION_ENGR;
//(* 
// * WP frame - origin at WP *
//  (if 3d have to first rotate at wp to get pitch and roll aligned with yaw arm)
// 1) translate origin to reference yaw pivot (translation)

// get coordinates as referenced from yaw pivot
X_OFFSETS[1] := X_OFFSET_BEGIN - YAW_ARM_LENGTH; 
Y_OFFSETS[1] := Y_OFFSET_BEGIN;

// * WP frame - origin at yaw pivot *
// 2) rotate origin at yaw pivot to match bs frame (rotation)
// YAW_ROTATION := AXES[AXIS_YAW].FEEDBACK.POSITION_ENGR; // offset from Boom Swing

// get coordinates as referenced from yaw pivot, along boom swing axis
X_OFFSETS[2] := X_OFFSETS[1] * COS_DEG(AXES[AXIS_YAW].FEEDBACK.POSITION_ENGR) - Y_OFFSETS[1] * SIN_DEG(AXES[AXIS_YAW].FEEDBACK.POSITION_ENGR); // rotate origin at yaw pivot by gps heading offset
Y_OFFSETS[2] := X_OFFSETS[1] * SIN_DEG(AXES[AXIS_YAW].FEEDBACK.POSITION_ENGR) + Y_OFFSETS[1] * COS_DEG(AXES[AXIS_YAW].FEEDBACK.POSITION_ENGR);

// * BS frame - origin AT yaw pivot *
// 3) translate origin to bs pivot

// get coordinates as referenced from boom swing pivot along boom swing axis
X_OFFSETS[3] := X_OFFSETS[2] - BS_PIVOT_TO_YAW_PIVOT;
Y_OFFSETS[3] := Y_OFFSETS[2];

// * BS frame - origin at BS pivot *
// 4) rotate origin at bs pivot to world frame
//	- rotate by BS_ANGLE_NS_DELTA
BS_ANGLE_NS_DELTA := YAW_OFFSET_BEGIN + -1 * AXES[AXIS_YAW].FEEDBACK.POSITION_ENGR; //(Yaw is opposite sign)
BS_ANGLE_WORLD_NS := BS_ANGLE_NS_DELTA + AXES[AXIS_BOOM_SWING].FEEDBACK.POSITION_ENGR;

// get coordinates as referenced from boom swing pivot along world North - South Line ( or point to point as set by gps system, typically NS )
X_OFFSETS[4] := X_OFFSETS[3] * COS_DEG(BS_ANGLE_NS_DELTA) - Y_OFFSETS[3] * SIN_DEG(BS_ANGLE_NS_DELTA); // rotate origin at yaw pivot by gps heading offset
Y_OFFSETS[4] := X_OFFSETS[3] * SIN_DEG(BS_ANGLE_NS_DELTA) + Y_OFFSETS[3] * COS_DEG(BS_ANGLE_NS_DELTA);

// * WORLD frame - origin at BS pivot *

// now use boom swing pivot as machine reference, as rwp targeting movement starts from it
// translate target ccordinates to greater of 1/3 of remaining distance or ALIGNMENT_TARGET

// get coordinates of approach to ALIGNMENT_TARGET in world frame referenced from BS pivot
Y_OFFSETS[5] := Y_OFFSETS[4]; // maintainig base of triangle to target
IF X_OFFSETS[4] > ALIGNMENT_TARGET THEN // bs pivot distance from target
	X_OFFSETS[5] := MAX(( X_OFFSETS[4] / 3 ), ALIGNMENT_TARGET);
ELSIF X_OFFSETS[4] < -ALIGNMENT_TARGET THEN
	X_OFFSETS[5] := MIN(( X_OFFSETS[4] / 3 ), -ALIGNMENT_TARGET);
ELSE
	// get world offsets in x and y from wp - now we just zero in on target
	//RotateGpsTdToWorldNS( X_TD := X_OFFSET_BEGIN, Y_TD := Y_OFFSET_BEGIN, YAW_BEGIN := YAW_OFFSET_BEGIN, 
	//					X_WORLD => X_OFFSETS[5], Y_WORLD => Y_OFFSETS[5] );
	X_OFFSETS[5] := X_OFFSETS[4] / 3;
END_IF

(*
IF X_OFFSETS[4] >= 0 THEN // bs pivot distance from target
	IF X_OFFSETS[4] > ( ALIGNMENT_TARGET + 20 ) THEN // start aligning as approach alignment_target
		X_OFFSETS[5] := MAX(( X_OFFSETS[4] / 3 ), ALIGNMENT_TARGET); // going forward, curve to ALIGNMENT_TARGET
	ELSE
		X_OFFSETS[5] := X_OFFSETS[4] / 3;
	END_IF
ELSE
	IF X_OFFSETS[4] < ( ALIGNMENT_TARGET - 120 ) THEN
		X_OFFSETS[5] := MIN(( X_OFFSETS[4] / 3 ), -ALIGNMENT_TARGET); // going backwards, curve to ALIGNMENT_TARGET
	ELSE
		X_OFFSETS[5] := X_OFFSETS[4] / 3;
	END_IF	
END_IF
Y_OFFSETS[5] := Y_OFFSETS[4];
*)

// get heading offset from North South line to new target
IF (X_OFFSETS[5] ) > 20 THEN // eliminate divide by zero when close
	HEADING_TO_TARGET := ATAN_DEG ( - Y_OFFSETS[5] / X_OFFSETS[5] );
ELSE
	HEADING_TO_TARGET := 0;
END_IF

// get heading offset from machine heading
HEADING_TO_TARGET_OFFSET := YAW_OFFSET_BEGIN + HEADING_TO_TARGET;
debug[30] := HEADING_TO_TARGET;
// drive tracks to head to new target

// reduce magnitude as approach target
//IF ABS ( X_OFFSET_BEGIN ) < 1 THEN
IF ABS ( GPS_AXES[GPS_X].OFFSET_WORLD_FRAME ) < 1 THEN

 	PROXIMITY_SLOWING_FACTOR := 0;
ELSE
 	PROXIMITY_SLOWING_FACTOR := MIN ( ( ( ABS( X_OFFSET_BEGIN )) / 10 ) , 1); // start slowing at 1m (offset already /10 above)
	debug[29] := PROXIMITY_SLOWING_FACTOR;
END_IF
REMOTE.LJ_LR := 100;
REMOTE.RJ_LR := 100;
MANUAL_SPEED_REDUCING_FACTOR := MAX ( ( ((( ABS(REMOTE.LJ_LR) + ABS(REMOTE.RJ_LR) ) / 2 ) - GPS_AUTO_TRACK_JOYSTICK_LIMIT ) / ( 100 - GPS_AUTO_TRACK_JOYSTICK_LIMIT ) ) , 0 ); 
debug[41] := MANUAL_SPEED_REDUCING_FACTOR;
LEFT_TRACK_OUTPUT := PROXIMITY_SLOWING_FACTOR * MAX (MIN ( ( - HEADING_TO_TARGET_OFFSET * 2 + 90), 100), -100); // limit to -100 < x < 100
debug[31] := LEFT_TRACK_OUTPUT;
IF LEFT_TRACK_OUTPUT < 0 THEN
	LEFT_TRACK_POSITIVE := FALSE;
ELSE
	LEFT_TRACK_POSITIVE := TRUE;
END_IF
RIGHT_TRACK_OUTPUT := PROXIMITY_SLOWING_FACTOR * MAX ( MIN ( HEADING_TO_TARGET_OFFSET * 2 + 90, 100), -100);// limit to 100
debug[32] := RIGHT_TRACK_OUTPUT;
IF RIGHT_TRACK_OUTPUT < 0 THEN
	RIGHT_TRACK_POSITIVE := FALSE;
ELSE
	RIGHT_TRACK_POSITIVE := TRUE;
END_IF

IF X_OFFSET_BEGIN >= 0 THEN // going forward, normal situation
	LEFT_TRACK_OUTPUT_MAGNITUDE:= TO_INT ( ABS( LEFT_TRACK_OUTPUT) );  // max 100
	LEFT_TRACK_OUTPUT_POSITIVE := LEFT_TRACK_POSITIVE;
	RIGHT_TRACK_OUTPUT_MAGNITUDE:= TO_INT ( ABS( RIGHT_TRACK_OUTPUT ) );  // max 100
	RIGHT_TRACK_OUTPUT_POSITIVE:= RIGHT_TRACK_POSITIVE;
ELSE // swap directions
	RIGHT_TRACK_OUTPUT_MAGNITUDE:= TO_INT ( ABS( LEFT_TRACK_OUTPUT ) );  // max 100
	RIGHT_TRACK_OUTPUT_POSITIVE := NOT(LEFT_TRACK_POSITIVE);
	LEFT_TRACK_OUTPUT_MAGNITUDE := TO_INT ( ABS( RIGHT_TRACK_OUTPUT ) );  // max 100
	LEFT_TRACK_OUTPUT_POSITIVE := NOT(RIGHT_TRACK_POSITIVE);
 END_IF

 (*
IF X_OFFSETS[5] >= 0 THEN
	AXES[AXIS_TRACK_LEFT].OUTPUT.MAGNITUDE := TO_WORD( ABS( LEFT_TRACK_OUTPUT ) * 10);  // max 1000
	AXES[AXIS_TRACK_LEFT].OUTPUT.POSITIVE := LEFT_TRACK_POSITIVE;
	AXES[AXIS_TRACK_RIGHT].OUTPUT.MAGNITUDE := TO_WORD( ABS( RIGHT_TRACK_OUTPUT ) * 10);  // max 1000
	AXES[AXIS_TRACK_RIGHT].OUTPUT.POSITIVE := RIGHT_TRACK_POSITIVE;
ELSE
	AXES[AXIS_TRACK_RIGHT].OUTPUT.MAGNITUDE := TO_WORD( ABS( LEFT_TRACK_OUTPUT ) * 10);  // max 1000
	AXES[AXIS_TRACK_RIGHT].OUTPUT.POSITIVE := NOT(LEFT_TRACK_POSITIVE);
	AXES[AXIS_TRACK_LEFT].OUTPUT.MAGNITUDE := TO_WORD( ABS( RIGHT_TRACK_OUTPUT ) * 10);  // max 1000
	AXES[AXIS_TRACK_LEFT].OUTPUT.POSITIVE := NOT(RIGHT_TRACK_POSITIVE);
 END_IF
*)

END_PROGRAM

// StandardPLC/Application/POUs/Utilities/Conversions/ByteArrayToText
FUNCTION ByteArrayToText : REAL // takes in array and returns a REAL

VAR_INPUT
	ARRAY_SIZE: INT := 4; // accept arrays of 2 - 8 BYTES
	LITTLE_ENDIAN: BOOL := TRUE;
	SIGNED_TWOS: BOOL := TRUE;
	SCALE: REAL;
	OFFSET: REAL;
	pUSINT: POINTER TO USINT; // must pass ADR() or will kill PLC
END_VAR

VAR_IN_OUT
	
END_VAR

VAR
	i: INT :=0;
	dataLWORD: LWORD :=0;
	PACK_ONES: BOOL := FALSE; // for signed 2's Complement to get negatives
END_VAR

(* Take in array of 4 BYTES and return a REAL
	1) combine BYTES into an LWORD
	2) scale and offset and return REAL

	Planned use is for de-serializing data where the  built-in conversion doesn't work
*)

IF (TO_SINT(pUSINT^)< 0) AND (NOT LITTLE_ENDIAN) AND SIGNED_TWOS THEN // negative number
	PACK_ONES := TRUE;
ELSE
	PACK_ONES := FALSE;
END_IF

dataLWORD := TO_LWORD(pUSINT^);
FOR i := 1 TO ARRAY_SIZE - 1 DO
	pUSINT := pUSINT + 1;
	IF LITTLE_ENDIAN THEN
		dataLWORD := dataLWORD + TO_LWORD(EXPT(256, i)) * TO_LWORD(pUSINT^);
	ELSE
		dataLWORD := dataLWORD * 256 + TO_LWORD(pUSINT^);
	END_IF
END_FOR

IF LITTLE_ENDIAN AND (TO_SINT(pUSINT^) < 0) THEN // negative number
	PACK_ONES := TRUE;
END_IF

IF PACK_ONES AND SIGNED_TWOS AND (ARRAY_SIZE < 8) THEN
	dataLWORD := dataLWORD + TO_LWORD(EXPT(256, i)) * TO_LWORD(-1);
END_IF

IF SIGNED_TWOS THEN
	ByteArrayToReal := TO_REAL(LWORD_TO_LINT(dataLWORD)) * SCALE + OFFSET;
ELSE
	ByteArrayToReal := TO_REAL(dataLWORD) * SCALE + OFFSET;
END_IF

END_FUNCTION

// StandardPLC/Application/POUs/Utilities/Conversions/ddt
FUNCTION ddt : REAL // returns new dx given desired rate of change and last x

VAR_INPUT
	TARGET_POS: REAL;
	TARGET_LAST: REAL; // IF initiating autofeedback move, send current position, else send last targeted position
	dxdt: REAL; // eg vel, or dv/dt acc
END_VAR
VAR
	LOOP_MAX_DELTA_P_PER_CYCLE: REAL;
	
	// testing var's
	CONTROL_FREQ_HZ: REAL := 50;
	
END_VAR


// maps desired max velocity to max position change / cycle
LOOP_MAX_DELTA_P_PER_CYCLE := dxdt / CONTROL_FREQ_HZ; // GPS_VEL deg / sec * 0.020 sec / cycle = GPS_LOOP_MAX deg / this cycle
	
IF ABS( TARGET_POS - TARGET_LAST ) > LOOP_MAX_DELTA_P_PER_CYCLE THEN	
	IF ( TARGET_POS - TARGET_LAST ) < 0 THEN // moving in (-) direction
		ddt := -1 * LOOP_MAX_DELTA_P_PER_CYCLE + TARGET_LAST; // limit position change to control velocity
	ELSE
		ddt := LOOP_MAX_DELTA_P_PER_CYCLE + TARGET_LAST;
	END_IF
ELSE
	ddt := TARGET_POS;
END_IF

(* 
notes: 
1) can be used to limit acceleration or jerk by layering upon itself
2) "To meet the criteria of a comfortable driving experience, the limit value for acceleration might reasonably be set to under 0.9 m/s2, and that of jerk to 0.6 m/s3"
  - Toward a Comfortable Driving Experience FOR a Self-Driving Shuttle Bus
  *)

END_FUNCTION

// StandardPLC/Application/POUs/Utilities/Conversions/ddt_max
FUNCTION ddt_max : REAL // returns new dx given desired rate of change and last x

VAR_INPUT
	TARGET_LAST: REAL; // IF initiating autofeedback move, send current position, else send last targeted position
	dxdt: REAL; // eg vel, or dv/dt acc, put in +/- depending on desired direction of move
END_VAR
VAR
	LOOP_MAX_DELTA_P_PER_CYCLE: REAL;
	
	// testing var's
	CONTROL_FREQ_HZ: REAL := 50;
	
END_VAR


// maps desired max velocity to max position change / cycle
LOOP_MAX_DELTA_P_PER_CYCLE := dxdt / CONTROL_FREQ_HZ; // GPS_VEL deg / sec * 0.020 sec / cycle = GPS_LOOP_MAX deg / this cycle
ddt_max := LOOP_MAX_DELTA_P_PER_CYCLE + TARGET_LAST;



(* 
notes: 
1) can be used to limit acceleration or jerk by layering upon itself, with final call being to ddt
2) "To meet the criteria of a comfortable driving experience, the limit value for acceleration might reasonably be set to under 0.9 m/s2, and that of jerk to 0.6 m/s3"
  - Toward a Comfortable Driving Experience FOR a Self-Driving Shuttle Bus
  *)

END_FUNCTION

// StandardPLC/Application/POUs/Utilities/Conversions/ddt_layers
FUNCTION_BLOCK ddt_layered_target// returns new dx given number of laers of ddt, initial position, and final position, up to 6 layers (pos, vel, acc, jerk, snap, crackle, pop)
VAR_IN_OUT
    ddt_limits : ARRAY[*] OF REAL; // ddt_limits[0] - pos limit, 1 - vel limit, 2 - acc limit, etc
END_VAR
VAR_INPUT
	TARGET_VALUE: REAL; // TRUE means value should be changing in positive direction
	TARGET_VALUE_LAST: REAL; // IF initiating autofeedback move, send current position, else send last targeted position
	NUM_DERIVATIVE_LAYERS: USINT := 1; // eg 1 - velocity, 2 - acceleration, 3 - jerk, 4 - snap, etc
	MAX_TOP_LAYER: REAL; // The maximum allowed value of the highest layer controlling value
END_VAR
VAR
	TARGETS: ARRAY [0..6] OF REAL := [7(0)]; // [1] - pos, [2] - velocity, etc
	TARGET_PRIORS: ARRAY [0..6] OF REAL := [7(0)];
	IS_POS: BOOL := TRUE;
	i: USINT := 0;
END_VAR

IF TARGET_VALUE = TARGET_VALUE_LAST THEN
	ddt_layered_target := TARGET_VALUE;
	RETURN;
END_IF

i := NUM_DERIVATIVE_LAYERS;
IS_POS := ((TARGET_VALUE - TARGET_VALUE_LAST) > 0);
TARGET_PRIORS[i] := MAX_TOP_LAYER;
WHILE i > 1 DO
	TARGET_VALUE[i] := ddt_max(IS_POS, TARGET_PRIORS[i], TARGET_PRIORS[i + 1]); 
		i := i - 1;
END_WHILE
	(*
TARGET_ACC := ddt_max(DELTA_IS_POS, LAST_ACC, MAXIMUM_JERK); // 10 deg/sec / control freg 50 cycle/sec // control jerk on initiation of track assist by limiting heading delta
LAST_ACC := TARGET_ACC;
// calculate max new vel allowed by new acc:
TARGET_VEL := ddt_max(DELTA_IS_POS, LAST_VEL, TARGET_ACC);
// calculate heading delta:
ddt_layered_target := ddt(HEADING_TO_TARGET_OFFSET, LAST_POS, TARGET_VEL); *)

(* 
notes: 
1) can be used to limit acceleration or jerk by layering upon itself, with final call being to ddt
2) "To meet the criteria of a comfortable driving experience, the limit value for acceleration might reasonably be set to under 0.9 m/s2, and that of jerk to 0.6 m/s3"
  - Toward a Comfortable Driving Experience FOR a Self-Driving Shuttle Bus
  *)

END_FUNCTION_BLOCK

// StandardPLC/Application/POUs/Utilities/ProfileGen/TrapezoidStart
FUNCTION TrapezoidStart : BOOL
VAR_INPUT
	pPROFILE: POINTER TO sTrapezoid;
	pSETPOINT: POINTER TO sSetpoint;
	TIME_NOW_US: DWORD;
	FB: sFeedback;
	POSITION_ENGR: REAL;
	VELOCITY_ENGR: REAL;
	ACCEL_ENGR: REAL;
END_VAR
VAR
	POSITION_RAW: DINT;
	VELOCITY_RAW: REAL;
	ACCEL_RAW: REAL;
	POSITION_DELTA: DINT;
	VMAX: REAL;
	ACCEL_TIME: DWORD;
	ACCEL_DISTANCE: DINT;
	CRUISE_DISTANCE: DINT;
	CRUISE_TIME: DWORD;
	V: REAL;
END_VAR

(* Convert user units to internal units, counts *)
POSITION_RAW := POS_ENGR_TO_RAW(FB, POSITION_ENGR);
VELOCITY_RAW := VEL_ENGR_TO_RAW(FB, VELOCITY_ENGR);
ACCEL_RAW := VEL_ENGR_TO_RAW(FB, ACCEL_ENGR);

pPROFILE^.POSITION_END := POSITION_RAW;
pPROFILE^.VELOCITY := VELOCITY_RAW;
pPROFILE^.ACCELERATION := ACCEL_RAW;

(* Is the move trapezoidal or triangular? *)
POSITION_DELTA := ABS(POSITION_RAW - FB.POSITION_RAW);
pPROFILE^.POSITION_START := FB.POSITION_RAW;

IF POSITION_DELTA <= TO_DINT(VELOCITY_RAW * VELOCITY_RAW / ACCEL_RAW) THEN
	(* Triangular move *)

	(* End of accel and end of cruise are at the same time *)
	VMAX := SQRT(DINT_TO_REAL(POSITION_DELTA) * ACCEL_RAW);
	ACCEL_TIME := REAL_TO_DWORD(1000000.0 * VMAX / ACCEL_RAW);

	pPROFILE^.TIME_ACCEL_END := TIME_NOW_US + ACCEL_TIME;
	pPROFILE^.TIME_CRUISE_END := pPROFILE^.TIME_ACCEL_END;
	pPROFILE^.TIME_DECEL_END := TIME_NOW_US + 2 * ACCEL_TIME;
	pPROFILE^.TIME_ACCEL := ACCEL_TIME;
	pPROFILE^.TIME_CRUISE := 0;
	pPROFILE^.TIME_DECEL := ACCEL_TIME;
ELSE
	(* Trapezoidal move *)
	ACCEL_TIME := REAL_TO_DWORD(1000000 * VELOCITY_RAW / ACCEL_RAW);
	ACCEL_DISTANCE := REAL_TO_DINT(VELOCITY_RAW * TO_REAL(ACCEL_TIME) / 2000000.0);
	CRUISE_DISTANCE := POSITION_DELTA - 2 * ACCEL_DISTANCE;
	CRUISE_TIME := REAL_TO_DWORD(1000000.0 * TO_REAL(CRUISE_DISTANCE) / VELOCITY_RAW);

	pPROFILE^.TIME_ACCEL_END := TIME_NOW_US + ACCEL_TIME;
	pPROFILE^.TIME_CRUISE_END := pPROFILE^.TIME_ACCEL_END + CRUISE_TIME;
	pPROFILE^.TIME_DECEL_END := pPROFILE^.TIME_CRUISE_END + ACCEL_TIME;
	pPROFILE^.TIME_ACCEL := ACCEL_TIME;
	pPROFILE^.TIME_CRUISE := CRUISE_TIME;
	pPROFILE^.TIME_DECEL := ACCEL_TIME;
END_IF;

IF POSITION_RAW > FB.POSITION_RAW THEN
	pPROFILE^.DIRECTION_POSITIVE := TRUE;
ELSE
	pPROFILE^.DIRECTION_POSITIVE := FALSE;
	pPROFILE^.ACCELERATION := -pPROFILE^.ACCELERATION;
	pPROFILE^.VELOCITY := -pPROFILE^.VELOCITY;
END_IF;

(* Initialize the structure that hold the setpoint *)
pSETPOINT^.VELOCITY_RAW := 0;
pSETPOINT^.POSITION_RAW := FB.POSITION_RAW;

pSETPOINT^.POSITION_ENGR := POSITION_ENGR;
pSETPOINT^.VELOCITY_ENGR := VELOCITY_ENGR;
pSETPOINT^.ACCELERATION_ENGR := ACCEL_ENGR;

pPROFILE^.TIME_SEGMENT_BEGIN := TIME_NOW_US;
pPROFILE^.POS_SEGMENT_BEGIN := FB.POSITION_RAW;
pPROFILE^.STATE := ACCEL;

END_FUNCTION

// StandardPLC/Application/POUs/Utilities/ProfileGen/TrapezoidStart_jerk
FUNCTION TrapezoidStart_jerk : BOOL
VAR_INPUT
	pPROFILE: POINTER TO sTrapezoid;
	pSETPOINT: POINTER TO sSetpoint;
	TIME_NOW_US: DWORD;
	FB: sFeedback;
	POSITION_ENGR: REAL;
	VELOCITY_ENGR: REAL;
	ACCEL_ENGR: REAL;
END_VAR
VAR
	POSITION_RAW: DINT;
	VELOCITY_RAW: REAL;
	ACCEL_RAW: REAL;
	POSITION_DELTA: DINT;
	VELOCITY_DELTA: DINT; //
	VMAX: REAL;
	JERK_TIME: DWORD; // half of accel_time
	ACCEL_TIME: DWORD;
	ACCEL_DISTANCE: DINT;
	CRUISE_DISTANCE: DINT;
	CRUISE_TIME: DWORD;
	V: REAL;
END_VAR

(*
with a given max jerk, max accel, max vel, and desired displacement, figure out profile that gets there fastest

if max velocity cannot be reached with given accel limits, then use one fourth of the distance to find the max accel ?

constant jerk equation for displacement: 
	s_f := s_o + v_o * t + 0.5 * a_o * t^2 + (j * t^3) / 6
	
	note: 	solve above for j * t^3  : 
			then use trapezoid or triangle to determine t with max accel and max vel.  
			Use that time to solve for j.  if starting from settled (v_o = 0 and a_o = 0) then j := 6 * (s_f - s_o) / t^3
			set this J for move
			calculate times
			
	
max jerk for given vel delta
	j_max = a_ss^2 / (v_f - v_o)
	
time to max accel:
	t_to_max_accel := (a_f - a_o) / j
time to max vel:
	t_to_max_vel := 2 * t_max_accel + ( (v_f - v_2) - (v_1 - v_o) / a_max )

move types:
if > 2 * t_to_max_vel >> smoothed trapezoid

elsif > 
	
*)

(* Convert user units to internal units, counts *)
POSITION_RAW := POS_ENGR_TO_RAW(FB, POSITION_ENGR);
VELOCITY_RAW := VEL_ENGR_TO_RAW(FB, VELOCITY_ENGR);
ACCEL_RAW := VEL_ENGR_TO_RAW(FB, ACCEL_ENGR);

pPROFILE^.POSITION_END := POSITION_RAW;
pPROFILE^.VELOCITY := VELOCITY_RAW;
pPROFILE^.ACCELERATION := ACCEL_RAW;

(* Is the move trapezoidal or triangular? *)
POSITION_DELTA := ABS(POSITION_RAW - FB.POSITION_RAW);
pPROFILE^.POSITION_START := FB.POSITION_RAW;

IF POSITION_DELTA <= TO_DINT(VELOCITY_RAW * VELOCITY_RAW / ACCEL_RAW) THEN
	(* Triangular move *)

	(* End of accel and end of cruise are at the same time *)
	VMAX := SQRT(DINT_TO_REAL(POSITION_DELTA) * ACCEL_RAW);
	ACCEL_TIME := REAL_TO_DWORD(1000000.0 * VMAX / ACCEL_RAW);
	CRUISE_TIME := 0;

	pPROFILE^.TIME_CRUISE := 0;
	pPROFILE^.TIME_DECEL := ACCEL_TIME;
	
ELSE
	(* Trapezoidal move *)
	ACCEL_TIME := REAL_TO_DWORD(1000000 * VELOCITY_RAW / ACCEL_RAW);
	ACCEL_DISTANCE := REAL_TO_DINT(VELOCITY_RAW * TO_REAL(ACCEL_TIME) / 2000000.0);
	CRUISE_DISTANCE := POSITION_DELTA - 2 * ACCEL_DISTANCE;
	CRUISE_TIME := REAL_TO_DWORD(1000000.0 * TO_REAL(CRUISE_DISTANCE) / VELOCITY_RAW);

	
	
END_IF;

(*	
	t_duration := 2 * ACCEL_TIME + CRUISE_TIME;
	j := 6 * (s_f - s_o) / t_duration^3
*)
pPROFILE^.TIME_ACCEL_END := TIME_NOW_US + ACCEL_TIME;
pPROFILE^.TIME_CRUISE_END := pPROFILE^.TIME_ACCEL_END + CRUISE_TIME;
pPROFILE^.TIME_DECEL_END := pPROFILE^.TIME_CRUISE_END + ACCEL_TIME;
pPROFILE^.TIME_CRUISE := CRUISE_TIME;
pPROFILE^.TIME_DECEL := ACCEL_TIME;
pPROFILE^.TIME_ACCEL := ACCEL_TIME;
// don't need to define these because can just use known values.  so don't have to modify sTrapezoid:
pPROFILE^.TIME_ACCEL_JERK_UP_END := pPROFILE^.TIME_ACCEL_END - (pPROFILE^.TIME_DECEL_END - pPROFILE^.TIME_CRUISE_END) / 2;
pPROFILE^.TIME_DECEL_JERK_DOWN_END := (pPROFILE^.TIME_CRUISE_END + pPROFILE^.TIME_DECEL_END) / 2;


IF POSITION_RAW > FB.POSITION_RAW THEN
	pPROFILE^.DIRECTION_POSITIVE := TRUE;
ELSE
	pPROFILE^.DIRECTION_POSITIVE := FALSE;
	pPROFILE^.ACCELERATION := -pPROFILE^.ACCELERATION;
	pPROFILE^.VELOCITY := -pPROFILE^.VELOCITY;
END_IF;

(* Initialize the structure that hold the setpoint *)
pSETPOINT^.VELOCITY_RAW := 0;
pSETPOINT^.POSITION_RAW := FB.POSITION_RAW;

pSETPOINT^.POSITION_ENGR := POSITION_ENGR;
pSETPOINT^.VELOCITY_ENGR := VELOCITY_ENGR;
pSETPOINT^.ACCELERATION_ENGR := ACCEL_ENGR;

pPROFILE^.TIME_SEGMENT_BEGIN := TIME_NOW_US;
pPROFILE^.POS_SEGMENT_BEGIN := FB.POSITION_RAW;
pPROFILE^.STATE := ACCEL;

END_FUNCTION

// StandardPLC/Application/POUs/GPS/GpsAxisIsNearTarget
FUNCTION GpsAxisIsNearTarget : BOOL
VAR_INPUT
	GPS_AXIS: INT;
	VEL_AND_OFFSET_SAME_SIGN: BOOL; // velocity sign to correct offset is same sign as offset
	NEARNESS_FACTOR: REAL;
END_VAR
VAR
	SIGN_SWITCHER: SINT;
END_VAR

GpsAxisIsNearTarget := FALSE;

IF VEL_AND_OFFSET_SAME_SIGN THEN
	SIGN_SWITCHER := 1;
ELSE
	SIGN_SWITCHER := -1;
END_IF

GpsAxisIsNearTarget := GPS_READY AND
							(ABS(GPS_AXES[GPS_AXIS].OFFSET) < GPS_AXES[GPS_AXIS].TARGET_LIMIT * NEARNESS_FACTOR) AND // on target
	 						( (AXES[GPS_AXIS].FEEDBACK.VELOCITY_ENGR * GPS_AXES[GPS_AXIS].OFFSET * TO_REAL(SIGN_SWITCHER)) >= 0 ) AND // stopped or moving towards 0 offset  
							(ABS(AXES[GPS_AXIS].FEEDBACK.VELOCITY_ENGR) < 0.1) // moving slowly - actuator default speeds range 3 - 4 
							;
// (* debug
debug[30 + GPS_AXIS] := (AXES[GPS_AXIS].FEEDBACK.VELOCITY_ENGR * GPS_AXES[GPS_AXIS].OFFSET * SIGN_SWITCHER); // *)
debug[40 + GPS_AXIS] := ABS(GPS_AXES[GPS_AXIS].OFFSET);
debug[60 + GPS_AXIS] := to_real(GpsAxisIsNearTarget);

END_FUNCTION

// StandardPLC/Application/POUs/GPS/GpsAxisIsOnTarget
FUNCTION GpsAxisIsOnTarget : BOOL
VAR_INPUT
	GPS_AXIS: INT;
	VEL_AND_OFFSET_SAME_SIGN: BOOL; // velocity sign to correct offset is same sign as offset
END_VAR
VAR
	SIGN_SWITCHER: SINT;
END_VAR

GpsAxisIsOnTarget := FALSE;

IF VEL_AND_OFFSET_SAME_SIGN THEN
	SIGN_SWITCHER := 1;
ELSE
	SIGN_SWITCHER := -1;
END_IF

GpsAxisIsOnTarget := 	GPS_READY AND
							ABS(GPS_AXES[GPS_AXIS].OFFSET) < GPS_AXES[GPS_AXIS].TARGET_LIMIT AND // on target
	 						((AXES[GPS_AXIS].FEEDBACK.VELOCITY_ENGR * GPS_AXES[GPS_AXIS].OFFSET) * SIGN_SWITCHER >= 0 ) AND // stopped or moving towards 0 offset  
							ABS(AXES[GPS_AXIS].FEEDBACK.VELOCITY_ENGR) < 0.05 // moving slowly - actuator default speeds range 3 - 4 
							;

END_FUNCTION

// StandardPLC/Application/Visualizations/GPS_RANGE
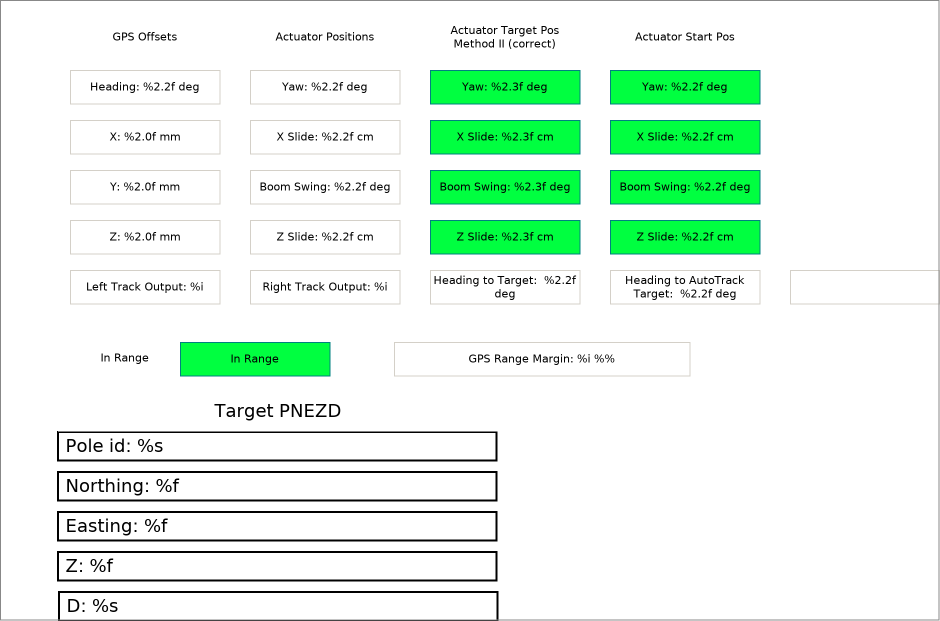
VISUALIZATION GPS_RANGE  // 940x621
    Label (50,343 150x30), "In Range"
    Textfield (180,342 150x34), "In Range", colour toggle: GPS_IN_RANGE[0] = 0
    Label (70,7 150x60), "GPS Offsets"
    Textfield (70,70 150x34), "Heading: %2.2f deg", text variable: GPS_SIM_OFFSETS[GPS_HEADING]
        OnMouseUp: write the text variable via Default
    Textfield (70,120 150x34), "X: %2.0f mm", text variable: GPS_SIM_OFFSETS[GPS_X]
        OnMouseUp: write the text variable via Default
    Textfield (70,170 150x34), "Y: %2.0f mm", text variable: GPS_SIM_OFFSETS[GPS_Y]
        OnMouseUp: write the text variable via Default
    Textfield (70,220 150x34), "Z: %2.0f mm", text variable: GPS_SIM_OFFSETS[GPS_Z]
        OnMouseUp: write the text variable via Default
    Label (250,7 150x60), "Actuator Positions"
    Textfield (250,70 150x34), "Yaw: %2.2f deg", text variable: AXES[AXIS_YAW].FEEDBACK.POSITION_ENGR
        OnMouseUp: write the text variable via Default
    Textfield (250,120 150x34), "X Slide: %2.2f cm", text variable: AXES[AXIS_X_SLIDE].FEEDBACK.POSITION_ENGR
        OnMouseUp: write the text variable via Default
    Textfield (250,170 150x34), "Boom Swing: %2.2f deg", text variable: AXES[AXIS_BOOM_SWING].FEEDBACK.POSITION_ENGR
        OnMouseUp: write the text variable via Default
    Textfield (250,220 150x34), "Z Slide: %2.2f cm", text variable: AXES[AXIS_Z_SLIDE].FEEDBACK.POSITION_ENGR
        OnMouseUp: write the text variable via Default
    Textfield (394,342 296x34), "GPS Range Margin: %i %%", text variable: GPS_RANGE_MARGIN
        OnMouseUp: write the text variable via Default
    Textfield (430,270 150x34), "Heading to Target: %2.2f deg", text variable: HEADING_TO_TARGET
    Label (610,7 150x60), "Actuator Start Pos"
    Textfield (610,70 150x34), "Yaw: %2.2f deg", text variable: AXES[AXIS_YAW].FEEDBACK.POSITION_ENGR, colour toggle: GPS_IN_RANGE[GPS_HEADING] = 0
        OnMouseUp: write the text variable via Default
    Textfield (610,120 150x34), "X Slide: %2.2f cm", text variable: AXES[AXIS_X_SLIDE].FEEDBACK.POSITION_ENGR, colour toggle: GPS_IN_RANGE[GPS_X] = 0
        OnMouseUp: write the text variable via Default
    Textfield (610,170 150x34), "Boom Swing: %2.2f deg", text variable: AXES[AXIS_BOOM_SWING].FEEDBACK.POSITION_ENGR, colour toggle: GPS_IN_RANGE[GPS_Y] = 0
        OnMouseUp: write the text variable via Default
    Textfield (610,220 150x34), "Z Slide: %2.2f cm", text variable: AXES[AXIS_Z_SLIDE].FEEDBACK.POSITION_ENGR, colour toggle: GPS_IN_RANGE[GPS_Z] = 0
        OnMouseUp: write the text variable via Default
    Label (430,7 150x60), "Actuator Target Pos Method II (correct)"
    Textfield (430,70 150x34), "Yaw: %2.3f deg", text variable: TARGET_POSITIONS_METHOD_2[GPS_HEADING], colour toggle: GPS_IN_RANGE[GPS_HEADING] = 0
        OnMouseUp: write the text variable via Default
    Textfield (430,120 150x34), "X Slide: %2.3f cm", text variable: TARGET_POSITIONS_METHOD_2[GPS_X], colour toggle: GPS_IN_RANGE[GPS_X] = 0
        OnMouseUp: write the text variable via Default
    Textfield (430,170 150x34), "Boom Swing: %2.3f deg", text variable: TARGET_POSITIONS_METHOD_2[GPS_Y], colour toggle: GPS_IN_RANGE[GPS_Y] = 0
        OnMouseUp: write the text variable via Default
    Textfield (430,220 150x34), "Z Slide: %2.3f cm", text variable: TARGET_POSITIONS_METHOD_2[GPS_Z], colour toggle: GPS_IN_RANGE[GPS_Z] = 0
        OnMouseUp: write the text variable via Default
    Textfield (790,270 150x34)
    Textfield (70,270 150x34), "Left Track Output: %i", text variable: LEFT_TRACK_OUTPUT
    Textfield (250,270 150x34), "Right Track Output: %i", text variable: RIGHT_TRACK_OUTPUT
    Rectangle (57,511 440x30), "Easting: %f", text variable: GPS_PNEZD_E
    Rectangle (57,471 440x30), "Northing: %f", text variable: GPS_PNEZD_N
    Rectangle (57,551 440x30), "Z: %f", text variable: GPS_PNEZD_Z
    Rectangle (57,431 440x30), "Pole id: %s", text variable: GPS_PNEZD_P
    Rectangle (58,591 440x30), "D: %s", text variable: GPS_PNEZD_D
    Rectangle (58,391 440x40), "Target PNEZD"
    Textfield (610,270 150x34), "Heading to AutoTrack Target: %2.2f deg", text variable: HEADING_TO_TARGET_OFFSET
END_VISUALIZATION

// StandardPLC/Application/Visualizations/FUNCTION_CHECK
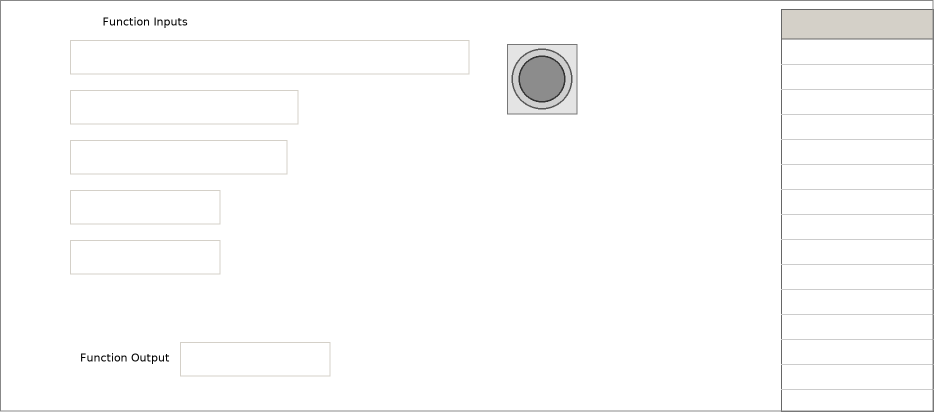
VISUALIZATION FUNCTION_CHECK  // 934x412
    Label (50,343 150x30), "Function Output"
    Textfield (180,342 150x34)
    Label (70,7 150x30), "Function Inputs"
    Textfield (70,40 399x34), text variable: GPS_PNEZD_D
        OnMouseUp: write the text variable via Edit
    Textfield (70,90 228x34)
    Textfield (70,140 217x34)
    Textfield (70,190 150x34)
    Textfield (70,240 150x34)
    PushSwitchLed (507,44 70x70), variable: Start_test, behaviour: TOGGLE, style: Switch-PushSwitchLed-Gray
    Table (781,9 153x403), data array: SCREW_COUNT
        p1014161805: Ojjo_TD.SCREW_LENGTHS_COUNT - 1 + 1
        p1098849879: 2 - 1 + 1
        p3854506369: SCREW_COUNT[1,INDEX]
        p1892666644: SCREW_COUNT[2,INDEX]
END_VISUALIZATION

// StandardPLC/Application/Visualizations/P_GPS_testing
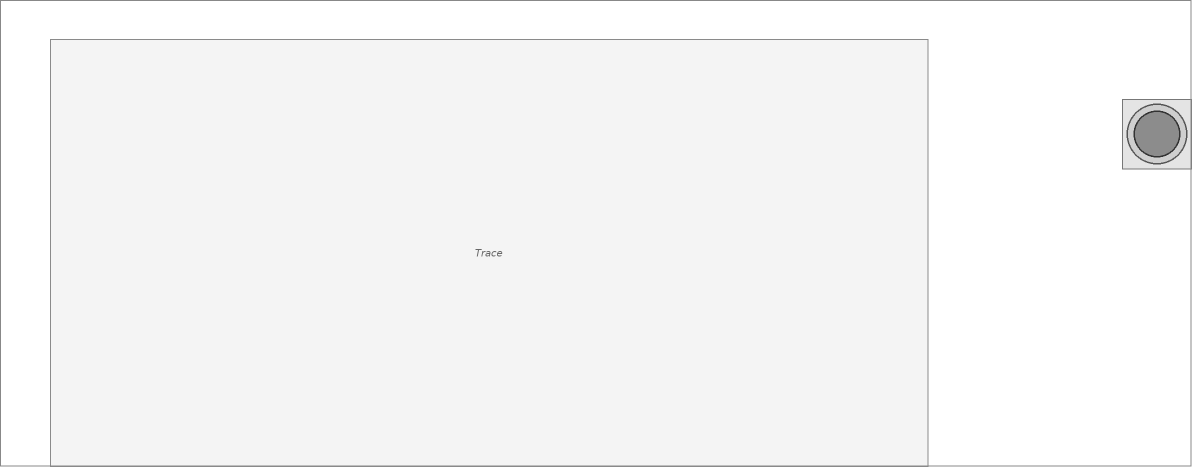
VISUALIZATION P_GPS_testing  // 1192x467
    Trace (50,39 878x428)
    PushSwitchLed (1122,99 70x70), variable: Start_test, behaviour: TOGGLE, style: Switch-PushSwitchLed-Gray
END_VISUALIZATION

// StandardPLC/Application/Visualizations/GRAPH_FUNCTION_RESULTS
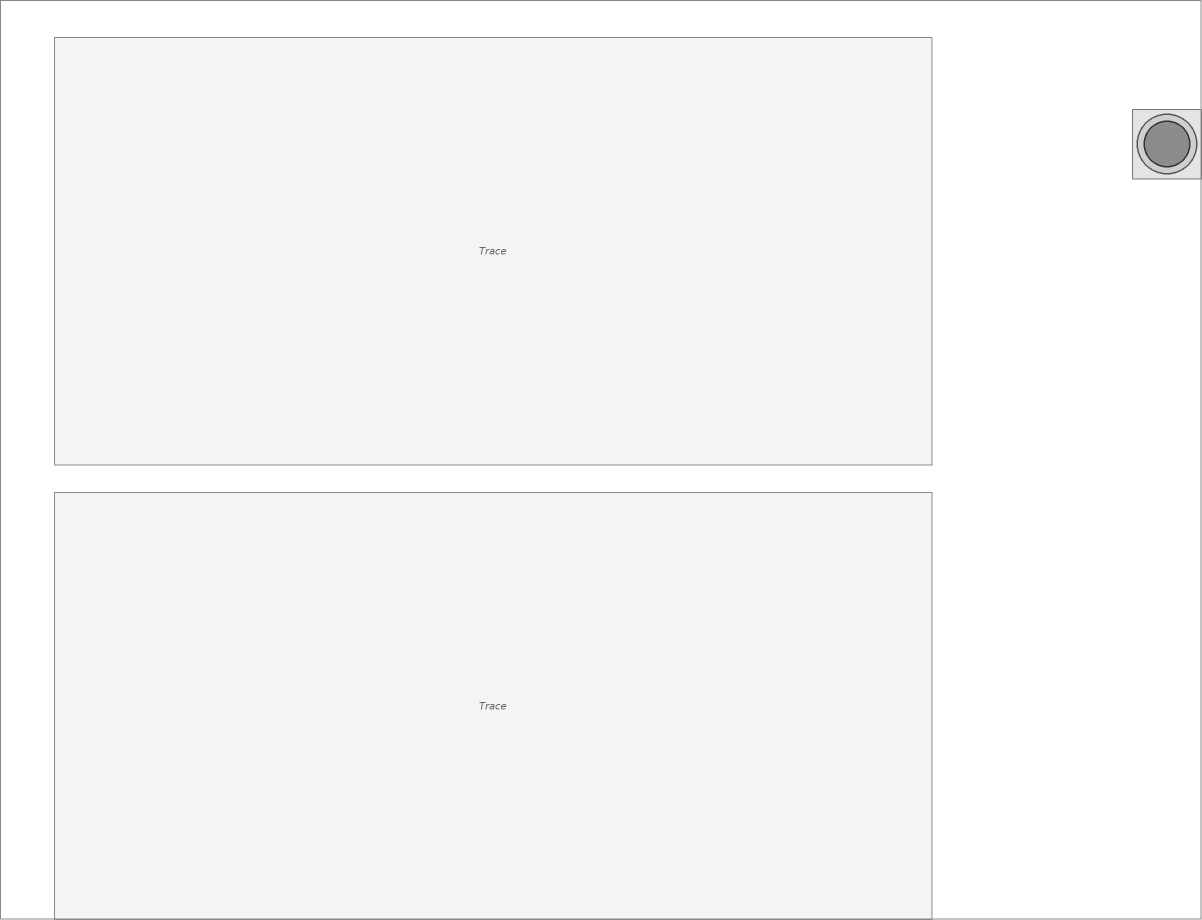
VISUALIZATION GRAPH_FUNCTION_RESULTS  // 1202x920
    Trace (54,37 878x428)
    PushSwitchLed (1132,109 70x70), variable: Start_test, behaviour: TOGGLE, style: Switch-PushSwitchLed-Gray
    Trace (54,492 878x428)
END_VISUALIZATION
